LIN {X 0.040,Y -180.708,Z 1755.470,A 0.000,B 0.000,C 90.000,E1 264.552} C_DIS
LIN {X -0.041,Y -178.793,Z 1755.442,A 0.000,B 0.000,C 90.000,E1 259.511} C_DIS
LIN {X 0.037,Y -175.839,Z 1755.413,A 0.000,B 0.000,C 90.000,E1 254.393} C_DIS
LIN {X 0.036,Y -172.030,Z 1755.385,A 0.000,B 0.000,C 90.000,E1 249.263} C_DIS
LIN {X 0.012,Y -171.457,Z 1755.380,A 0.000,B 0.000,C 90.000,E1 248.411} C_DIS
LIN {X -0.008,Y -167.690,Z 1755.356,A 0.000,B 0.000,C 90.000,E1 244.101} C_DIS
LIN {X 0.006,Y -166.372,Z 1755.346,A 0.000,B 0.000,C 90.000,E1 242.359} C_DIS
LIN {X -0.001,Y -163.102,Z 1755.327,A 0.000,B 0.000,C 90.000,E1 238.869} C_DIS
LIN {X 0.048,Y -161.048,Z 1755.312,A 0.000,B 0.000,C 90.000,E1 236.215} C_DIS
LIN {X 0.033,Y -157.785,Z 1755.293,A 0.000,B 0.000,C 90.000,E1 232.683} C_DIS
LIN {X -0.024,Y -155.821,Z 1755.278,A 0.000,B 0.000,C 90.000,E1 230.033} C_DIS
LIN {X -0.067,Y -152.073,Z 1755.253,A 0.000,B 0.000,C 90.000,E1 225.567} C_DIS
LIN {X -0.048,Y -150.322,Z 1755.238,A 0.000,B 0.000,C 90.000,E1 222.852} C_DIS
LIN {X -0.026,Y -147.065,Z 1755.213,A 0.000,B 0.000,C 90.000,E1 218.302} C_DIS
LIN {X 0.081,Y -145.640,Z 1755.198,A 0.000,B 0.000,C 90.000,E1 215.518} C_DIS
LIN {X 0.079,Y -143.023,Z 1755.172,A 0.000,B 0.000,C 90.000,E1 210.924} C_DIS
LIN {X 0.010,Y -141.649,Z 1755.151,A 0.000,B 0.000,C 90.000,E1 207.257} C_DIS
LIN {X 0.060,Y -139.443,Z 1755.115,A 0.000,B 0.000,C 90.000,E1 200.737} C_DIS
LIN {X -0.018,Y -139.175,Z 1755.105,A 0.000,B 0.000,C 90.000,E1 198.906} C_DIS
LIN {X 0.010,Y -138.319,Z 1755.053,A 0.000,B 0.000,C 90.000,E1 189.557} C_DIS
LIN {X 0.019,Y -139.469,Z 1755.006,A 0.000,B 0.000,C 90.000,E1 181.146} C_DIS
LIN {X -0.040,Y -141.038,Z 1754.975,A 0.000,B 0.000,C 90.000,E1 175.584} C_DIS
LIN {X 0.055,Y -142.406,Z 1754.960,A 0.000,B 0.000,C 90.000,E1 172.761} C_DIS
LIN {X -0.024,Y -144.639,Z 1754.934,A 0.000,B 0.000,C 90.000,E1 168.173} C_DIS
LIN {X 0.036,Y -147.835,Z 1754.909,A 0.000,B 0.000,C 90.000,E1 163.559} C_DIS
LIN {X -0.020,Y -150.531,Z 1754.888,A 0.000,B 0.000,C 90.000,E1 159.934} C_DIS
LIN {X -0.001,Y -153.994,Z 1754.868,A 0.000,B 0.000,C 90.000,E1 156.305} C_DIS
LIN {X -0.080,Y -157.408,Z 1754.848,A 0.000,B 0.000,C 90.000,E1 152.743} C_DIS
LIN {X -0.001,Y -161.616,Z 1754.829,A 0.000,B 0.000,C 90.000,E1 149.154} C_DIS
LIN {X 0.101,Y -165.813,Z 1754.809,A 0.000,B 0.000,C 90.000,E1 145.595} C_DIS
LIN {X -0.011,Y -170.780,Z 1754.790,A 0.000,B 0.000,C 90.000,E1 142.145} C_DIS
LIN {X 0.012,Y -175.651,Z 1754.771,A 0.000,B 0.000,C 90.000,E1 138.690} C_DIS
LIN {X 0.009,Y -181.266,Z 1754.752,A 0.000,B 0.000,C 90.000,E1 135.283} C_DIS
LIN {X 0.009,Y -186.740,Z 1754.733,A 0.000,B 0.000,C 90.000,E1 131.919} C_DIS
LIN {X -0.039,Y -191.336,Z 1754.719,A 0.000,B 0.000,C 90.000,E1 129.439} C_DIS
LIN {X 0.007,Y -197.170,Z 1754.701,A 0.000,B 0.000,C 90.000,E1 126.137} C_DIS
LIN {X -0.075,Y -200.448,Z 1754.692,A 0.000,B 0.000,C 90.000,E1 124.532} C_DIS
LIN {X 0.108,Y -206.331,Z 1754.674,A 0.000,B 0.000,C 90.000,E1 121.258} C_DIS
LIN {X 0.076,Y -210.527,Z 1754.662,A 0.000,B 0.000,C 90.000,E1 119.205} C_DIS
LIN {X 0.072,Y -336.076,Z 1754.662,A 0.000,B 0.000,C 90.000,E1 119.205} C_DIS
LIN {X -0.025,Y -337.451,Z 1754.662,A 0.000,B 0.000,C 90.000,E1 119.205} C_DIS
LIN {X -0.160,Y -341.637,Z 1754.661,A 0.000,B 0.000,C 90.000,E1 119.077} C_DIS
LIN {X 0.005,Y -343.914,Z 1754.661,A 0.000,B 0.000,C 90.000,E1 118.899} C_DIS
LIN {X 0.117,Y -347.777,Z 1754.658,A 0.000,B 0.000,C 90.000,E1 118.487} C_DIS
LIN {X -0.014,Y -349.661,Z 1754.657,A 0.000,B 0.000,C 90.000,E1 118.231} C_DIS
LIN {X 0.039,Y -352.528,Z 1754.654,A 0.000,B 0.000,C 90.000,E1 117.641} C_DIS
LIN {X -0.051,Y -365.817,Z 1754.639,A 0.000,B 0.000,C 90.000,E1 114.951} C_DIS
LIN {X 0.124,Y -380.655,Z 1754.624,A 0.000,B 0.000,C 90.000,E1 112.280} C_DIS
LIN {X 0.058,Y -395.252,Z 1754.611,A 0.000,B 0.000,C 90.000,E1 109.993} C_DIS
LIN {X -0.057,Y -411.275,Z 1754.599,A 0.000,B 0.000,C 90.000,E1 107.764} C_DIS
LIN {X 0.109,Y -428.838,Z 1754.586,A 0.000,B 0.000,C 90.000,E1 105.552} C_DIS
LIN {X 0.213,Y -448.012,Z 1754.575,A 0.000,B 0.000,C 90.000,E1 103.411} C_DIS
LIN {X -0.213,Y -468.079,Z 1754.564,A 0.000,B 0.000,C 90.000,E1 101.478} C_DIS
LIN {X 0.253,Y -491.305,Z 1754.552,A 0.000,B 0.000,C 90.000,E1 99.378} C_DIS
LIN {X -0.047,Y -509.698,Z 1754.544,A 0.000,B 0.000,C 90.000,E1 97.936} C_DIS
LIN {X 0.195,Y -512.101,Z 1754.543,A 0.000,B 0.000,C 90.000,E1 97.701} C_DIS
LIN {X -0.240,Y -513.995,Z 1754.542,A 0.000,B 0.000,C 90.000,E1 97.530} C_DIS
LIN {X -0.100,Y -515.433,Z 1754.541,A 0.000,B 0.000,C 90.000,E1 97.296} C_DIS
LIN {X -0.240,Y -517.449,Z 1754.538,A 0.000,B 0.000,C 90.000,E1 96.834} C_DIS
LIN {X 0.143,Y -518.273,Z 1754.535,A 0.000,B 0.000,C 90.000,E1 96.315} C_DIS
LIN {X 0.022,Y -518.062,Z 1754.532,A 0.000,B 0.000,C 90.000,E1 95.853} C_DIS
LIN {X -0.097,Y -516.785,Z 1754.530,A 0.000,B 0.000,C 90.000,E1 95.391} C_DIS
LIN {X -0.179,Y -515.682,Z 1754.529,A 0.000,B 0.000,C 90.000,E1 95.163} C_DIS
LIN {X 0.206,Y -512.472,Z 1754.526,A 0.000,B 0.000,C 90.000,E1 94.645} C_DIS
LIN {X -0.042,Y -498.764,Z 1754.515,A 0.000,B 0.000,C 90.000,E1 92.751} C_DIS
LIN {X -0.166,Y -489.865,Z 1754.509,A 0.000,B 0.000,C 90.000,E1 91.547} C_DIS
LIN {X 0.038,Y -475.234,Z 1754.497,A 0.000,B 0.000,C 90.000,E1 89.542} C_DIS
LIN {X -0.133,Y -464.235,Z 1754.489,A 0.000,B 0.000,C 90.000,E1 88.051} C_DIS
LIN {X -0.045,Y -449.558,Z 1754.478,A 0.000,B 0.000,C 90.000,E1 85.988} C_DIS
LIN {X 0.029,Y -436.773,Z 1754.468,A 0.000,B 0.000,C 90.000,E1 84.147} C_DIS
LIN {X 0.170,Y -420.678,Z 1754.454,A 0.000,B 0.000,C 90.000,E1 81.724} C_DIS
LIN {X 0.111,Y -403.545,Z 1754.439,A 0.000,B 0.000,C 90.000,E1 78.993} C_DIS
LIN {X 0.190,Y -387.313,Z 1754.423,A 0.000,B 0.000,C 90.000,E1 76.172} C_DIS
LIN {X -0.120,Y -374.927,Z 1754.411,A 0.000,B 0.000,C 90.000,E1 73.921} C_DIS
LIN {X -0.149,Y -362.921,Z 1754.398,A 0.000,B 0.000,C 90.000,E1 71.583} C_DIS
LIN {X 0.096,Y -351.274,Z 1754.384,A 0.000,B 0.000,C 90.000,E1 69.156} C_DIS
LIN {X 0.118,Y -337.342,Z 1754.367,A 0.000,B 0.000,C 90.000,E1 66.102} C_DIS
LIN {X -0.021,Y -327.838,Z 1754.355,A 0.000,B 0.000,C 90.000,E1 63.948} C_DIS
LIN {X 0.149,Y -317.156,Z 1754.341,A 0.000,B 0.000,C 90.000,E1 61.385} C_DIS
LIN {X 0.069,Y -310.275,Z 1754.332,A 0.000,B 0.000,C 90.000,E1 59.793} C_DIS
LIN {X -0.116,Y -303.074,Z 1754.323,A 0.000,B 0.000,C 90.000,E1 58.201} C_DIS
LIN {X 0.091,Y -291.430,Z 1754.308,A 0.000,B 0.000,C 90.000,E1 55.515} C_DIS
LIN {X -0.022,Y -281.370,Z 1754.295,A 0.000,B 0.000,C 90.000,E1 53.176} C_DIS
LIN {X -0.088,Y -270.159,Z 1754.280,A 0.000,B 0.000,C 90.000,E1 50.436} C_DIS
LIN {X -0.127,Y -259.442,Z 1754.265,A 0.000,B 0.000,C 90.000,E1 47.634} C_DIS
LIN {X -0.123,Y -251.556,Z 1754.253,A 0.000,B 0.000,C 90.000,E1 45.486} C_DIS
LIN {X 0.050,Y -240.177,Z 1754.234,A 0.000,B 0.000,C 90.000,E1 42.162} C_DIS
LIN {X -0.059,Y -229.392,Z 1754.216,A 0.000,B 0.000,C 90.000,E1 38.830} C_DIS
LIN {X 0.037,Y -220.401,Z 1754.199,A 0.000,B 0.000,C 90.000,E1 35.758} C_DIS
LIN {X -0.010,Y -214.074,Z 1754.186,A 0.000,B 0.000,C 90.000,E1 33.452} C_DIS
LIN {X -0.091,Y -206.447,Z 1754.168,A 0.000,B 0.000,C 90.000,E1 30.335} C_DIS
LIN {X -0.035,Y -199.500,Z 1754.151,A 0.000,B 0.000,C 90.000,E1 27.129} C_DIS
LIN {X -0.065,Y -193.231,Z 1754.133,A 0.000,B 0.000,C 90.000,E1 23.898} C_DIS
LIN {X -0.047,Y -187.807,Z 1754.114,A 0.000,B 0.000,C 90.000,E1 20.610} C_DIS
LIN {X -0.012,Y -183.120,Z 1754.096,A 0.000,B 0.000,C 90.000,E1 17.275} C_DIS
LIN {X 0.093,Y -179.345,Z 1754.077,A 0.000,B 0.000,C 90.000,E1 13.883} C_DIS
LIN {X 0.020,Y -175.766,Z 1754.054,A 0.000,B 0.000,C 90.000,E1 9.670} C_DIS
LIN {X 0.052,Y -172.721,Z 1754.025,A 0.000,B 0.000,C 90.000,E1 4.531} C_DIS
LIN {X -0.052,Y -171.069,Z 1753.983,A 0.000,B 0.000,C 90.000,E1 356.963} C_DIS
LIN {X -0.058,Y -171.916,Z 1753.935,A 0.000,B 0.000,C 90.000,E1 348.342} C_DIS
LIN {X -0.011,Y -174.125,Z 1753.902,A 0.000,B 0.000,C 90.000,E1 342.308} C_DIS
LIN {X -0.005,Y -177.557,Z 1753.873,A 0.000,B 0.000,C 90.000,E1 337.177} C_DIS
LIN {X 0.041,Y -181.260,Z 1753.850,A 0.000,B 0.000,C 90.000,E1 332.922} C_DIS
LIN {X -0.056,Y -184.980,Z 1753.831,A 0.000,B 0.000,C 90.000,E1 329.587} C_DIS
LIN {X 0.061,Y -189.516,Z 1753.812,A 0.000,B 0.000,C 90.000,E1 326.215} C_DIS
LIN {X 0.027,Y -195.012,Z 1753.794,A 0.000,B 0.000,C 90.000,E1 322.924} C_DIS
LIN {X 0.007,Y -199.781,Z 1753.781,A 0.000,B 0.000,C 90.000,E1 320.481} C_DIS
LIN {X 0.088,Y -206.288,Z 1753.765,A 0.000,B 0.000,C 90.000,E1 317.634} C_DIS
LIN {X 0.112,Y -212.607,Z 1753.751,A 0.000,B 0.000,C 90.000,E1 315.243} C_DIS
LIN {X 0.048,Y -218.582,Z 1753.741,A 0.000,B 0.000,C 90.000,E1 313.299} C_DIS
LIN {X -0.061,Y -225.378,Z 1753.730,A 0.000,B 0.000,C 90.000,E1 311.391} C_DIS
LIN {X -0.016,Y -231.515,Z 1753.721,A 0.000,B 0.000,C 90.000,E1 309.850} C_DIS
LIN {X -0.007,Y -238.420,Z 1753.713,A 0.000,B 0.000,C 90.000,E1 308.338} C_DIS
LIN {X 0.089,Y -250.033,Z 1753.701,A 0.000,B 0.000,C 90.000,E1 306.091} C_DIS
LIN {X 0.078,Y -260.616,Z 1753.691,A 0.000,B 0.000,C 90.000,E1 304.278} C_DIS
LIN {X 0.027,Y -279.018,Z 1753.675,A 0.000,B 0.000,C 90.000,E1 301.465} C_DIS
LIN {X 0.018,Y -296.314,Z 1753.661,A 0.000,B 0.000,C 90.000,E1 299.077} C_DIS
LIN {X 0.108,Y -314.364,Z 1753.649,A 0.000,B 0.000,C 90.000,E1 296.744} C_DIS
LIN {X -0.008,Y -330.250,Z 1753.638,A 0.000,B 0.000,C 90.000,E1 294.847} C_DIS
LIN {X 0.141,Y -343.384,Z 1753.629,A 0.000,B 0.000,C 90.000,E1 293.259} C_DIS
LIN {X -0.111,Y -356.226,Z 1753.621,A 0.000,B 0.000,C 90.000,E1 291.770} C_DIS
LIN {X -0.037,Y -366.016,Z 1753.614,A 0.000,B 0.000,C 90.000,E1 290.556} C_DIS
LIN {X 0.204,Y -372.830,Z 1753.609,A 0.000,B 0.000,C 90.000,E1 289.631} C_DIS
LIN {X 0.024,Y -378.910,Z 1753.604,A 0.000,B 0.000,C 90.000,E1 288.779} C_DIS
LIN {X 0.136,Y -382.533,Z 1753.601,A 0.000,B 0.000,C 90.000,E1 288.181} C_DIS
LIN {X -0.091,Y -385.669,Z 1753.598,A 0.000,B 0.000,C 90.000,E1 287.638} C_DIS
LIN {X 0.069,Y -388.324,Z 1753.595,A 0.000,B 0.000,C 90.000,E1 287.040} C_DIS
LIN {X -0.124,Y -390.623,Z 1753.592,A 0.000,B 0.000,C 90.000,E1 286.496} C_DIS
LIN {X 0.070,Y -392.522,Z 1753.588,A 0.000,B 0.000,C 90.000,E1 285.898} C_DIS
LIN {X -0.215,Y -394.106,Z 1753.585,A 0.000,B 0.000,C 90.000,E1 285.371} C_DIS
LIN {X -0.002,Y -395.323,Z 1753.582,A 0.000,B 0.000,C 90.000,E1 284.773} C_DIS
LIN {X 0.123,Y -396.187,Z 1753.579,A 0.000,B 0.000,C 90.000,E1 284.189} C_DIS
LIN {X -0.034,Y -396.671,Z 1753.576,A 0.000,B 0.000,C 90.000,E1 283.647} C_DIS
LIN {X 0.105,Y -396.800,Z 1753.573,A 0.000,B 0.000,C 90.000,E1 283.063} C_DIS
LIN {X -0.138,Y -396.538,Z 1753.570,A 0.000,B 0.000,C 90.000,E1 282.535} C_DIS
LIN {X 0.008,Y -395.863,Z 1753.566,A 0.000,B 0.000,C 90.000,E1 281.951} C_DIS
LIN {X 0.152,Y -394.688,Z 1753.563,A 0.000,B 0.000,C 90.000,E1 281.366} C_DIS
LIN {X -0.095,Y -393.020,Z 1753.560,A 0.000,B 0.000,C 90.000,E1 280.838} C_DIS
LIN {X 0.037,Y -390.808,Z 1753.557,A 0.000,B 0.000,C 90.000,E1 280.254} C_DIS
LIN {X 0.149,Y -388.030,Z 1753.554,A 0.000,B 0.000,C 90.000,E1 279.670} C_DIS
LIN {X -0.037,Y -380.278,Z 1753.546,A 0.000,B 0.000,C 90.000,E1 278.276} C_DIS
LIN {X 0.025,Y -375.925,Z 1753.541,A 0.000,B 0.000,C 90.000,E1 277.409} C_DIS
LIN {X -0.008,Y -372.510,Z 1753.538,A 0.000,B 0.000,C 90.000,E1 276.834} C_DIS
LIN {X -0.058,Y -368.487,Z 1753.535,A 0.000,B 0.000,C 90.000,E1 276.258} C_DIS
LIN {X -0.127,Y -363.774,Z 1753.531,A 0.000,B 0.000,C 90.000,E1 275.682} C_DIS
LIN {X 0.136,Y -358.283,Z 1753.528,A 0.000,B 0.000,C 90.000,E1 275.049} C_DIS
LIN {X -0.072,Y -352.446,Z 1753.525,A 0.000,B 0.000,C 90.000,E1 274.531} C_DIS
LIN {X -0.027,Y -346.500,Z 1753.522,A 0.000,B 0.000,C 90.000,E1 274.012} C_DIS
LIN {X 0.160,Y -340.378,Z 1753.520,A 0.000,B 0.000,C 90.000,E1 273.498} C_DIS
LIN {X 0.024,Y -330.914,Z 1753.516,A 0.000,B 0.000,C 90.000,E1 272.865} C_DIS
LIN {X 0.057,Y -324.422,Z 1753.514,A 0.000,B 0.000,C 90.000,E1 272.465} C_DIS
LIN {X -0.040,Y -317.608,Z 1753.512,A 0.000,B 0.000,C 90.000,E1 272.121} C_DIS
LIN {X 0.117,Y -310.610,Z 1753.510,A 0.000,B 0.000,C 90.000,E1 271.776} C_DIS
LIN {X -0.078,Y -303.341,Z 1753.509,A 0.000,B 0.000,C 90.000,E1 271.547} C_DIS
LIN {X 0.069,Y -292.260,Z 1753.507,A 0.000,B 0.000,C 90.000,E1 271.203} C_DIS
LIN {X 0.001,Y -281.588,Z 1753.505,A 0.000,B 0.000,C 90.000,E1 270.974} C_DIS
LIN {X -0.106,Y -273.354,Z 1753.505,A 0.000,B 0.000,C 90.000,E1 270.859} C_DIS
LIN {X -0.092,Y -258.515,Z 1753.504,A 0.000,B 0.000,C 90.000,E1 270.688} C_DIS
LIN {X 0.031,Y -239.967,Z 1753.503,A 0.000,B 0.000,C 90.000,E1 270.516} C_DIS
LIN {X -0.015,Y -237.145,Z 1753.503,A 0.000,B 0.000,C 90.000,E1 270.516} C_DIS
LIN {X -0.047,Y -181.565,Z 1753.503,A 0.000,B 0.000,C 90.000,E1 270.516} C_DIS
LIN {X 0.054,Y -181.117,Z 1753.489,A 0.000,B 0.000,C 90.000,E1 267.936} C_DIS
LIN {X 0.042,Y -180.906,Z 1753.475,A 0.000,B 0.000,C 90.000,E1 265.412} C_DIS
LIN {X -0.081,Y -180.716,Z 1753.470,A 0.000,B 0.000,C 90.000,E1 264.609} C_DIS
LIN {X 0.017,Y -178.804,Z 1753.442,A 0.000,B 0.000,C 90.000,E1 259.511} C_DIS
LIN {X 0.093,Y -175.848,Z 1753.413,A 0.000,B 0.000,C 90.000,E1 254.393} C_DIS
LIN {X 0.053,Y -172.584,Z 1753.390,A 0.000,B 0.000,C 90.000,E1 250.134} C_DIS
LIN {X 0.069,Y -171.474,Z 1753.380,A 0.000,B 0.000,C 90.000,E1 248.411} C_DIS
LIN {X 0.048,Y -167.704,Z 1753.356,A 0.000,B 0.000,C 90.000,E1 244.101} C_DIS
LIN {X 0.061,Y -166.391,Z 1753.347,A 0.000,B 0.000,C 90.000,E1 242.359} C_DIS
LIN {X 0.052,Y -163.118,Z 1753.327,A 0.000,B 0.000,C 90.000,E1 238.869} C_DIS
LIN {X 0.102,Y -161.067,Z 1753.313,A 0.000,B 0.000,C 90.000,E1 236.215} C_DIS
LIN {X -0.010,Y -157.800,Z 1753.293,A 0.000,B 0.000,C 90.000,E1 232.718} C_DIS
LIN {X -0.072,Y -155.836,Z 1753.278,A 0.000,B 0.000,C 90.000,E1 230.070} C_DIS
LIN {X -0.015,Y -152.086,Z 1753.253,A 0.000,B 0.000,C 90.000,E1 225.567} C_DIS
LIN {X 0.004,Y -150.337,Z 1753.238,A 0.000,B 0.000,C 90.000,E1 222.852} C_DIS
LIN {X 0.025,Y -147.076,Z 1753.213,A 0.000,B 0.000,C 90.000,E1 218.302} C_DIS
LIN {X -0.071,Y -145.650,Z 1753.198,A 0.000,B 0.000,C 90.000,E1 215.598} C_DIS
LIN {X -0.067,Y -143.032,Z 1753.172,A 0.000,B 0.000,C 90.000,E1 211.003} C_DIS
LIN {X 0.059,Y -141.657,Z 1753.152,A 0.000,B 0.000,C 90.000,E1 207.257} C_DIS
LIN {X -0.022,Y -139.447,Z 1753.115,A 0.000,B 0.000,C 90.000,E1 200.791} C_DIS
LIN {X 0.031,Y -139.180,Z 1753.105,A 0.000,B 0.000,C 90.000,E1 198.906} C_DIS
LIN {X 0.059,Y -138.320,Z 1753.053,A 0.000,B 0.000,C 90.000,E1 189.557} C_DIS
LIN {X 0.069,Y -139.465,Z 1753.006,A 0.000,B 0.000,C 90.000,E1 181.146} C_DIS
LIN {X 0.010,Y -141.029,Z 1752.975,A 0.000,B 0.000,C 90.000,E1 175.584} C_DIS
LIN {X -0.036,Y -142.396,Z 1752.960,A 0.000,B 0.000,C 90.000,E1 172.818} C_DIS
LIN {X 0.026,Y -144.628,Z 1752.934,A 0.000,B 0.000,C 90.000,E1 168.173} C_DIS
LIN {X -0.055,Y -147.823,Z 1752.909,A 0.000,B 0.000,C 90.000,E1 163.614} C_DIS
LIN {X 0.031,Y -150.514,Z 1752.889,A 0.000,B 0.000,C 90.000,E1 159.934} C_DIS
LIN {X 0.052,Y -153.976,Z 1752.868,A 0.000,B 0.000,C 90.000,E1 156.305} C_DIS
LIN {X -0.027,Y -157.387,Z 1752.849,A 0.000,B 0.000,C 90.000,E1 152.743} C_DIS
LIN {X -0.085,Y -161.592,Z 1752.829,A 0.000,B 0.000,C 90.000,E1 149.203} C_DIS
LIN {X -0.075,Y -165.789,Z 1752.809,A 0.000,B 0.000,C 90.000,E1 145.674} C_DIS
LIN {X -0.089,Y -170.750,Z 1752.790,A 0.000,B 0.000,C 90.000,E1 142.190} C_DIS
LIN {X 0.069,Y -175.622,Z 1752.771,A 0.000,B 0.000,C 90.000,E1 138.690} C_DIS
LIN {X -0.062,Y -181.238,Z 1752.752,A 0.000,B 0.000,C 90.000,E1 135.324} C_DIS
LIN {X 0.069,Y -186.708,Z 1752.733,A 0.000,B 0.000,C 90.000,E1 131.919} C_DIS
LIN {X 0.021,Y -191.307,Z 1752.719,A 0.000,B 0.000,C 90.000,E1 129.439} C_DIS
LIN {X -0.048,Y -197.136,Z 1752.701,A 0.000,B 0.000,C 90.000,E1 126.171} C_DIS
LIN {X -0.013,Y -200.413,Z 1752.692,A 0.000,B 0.000,C 90.000,E1 124.532} C_DIS
LIN {X -0.112,Y -206.297,Z 1752.674,A 0.000,B 0.000,C 90.000,E1 121.337} C_DIS
LIN {X -0.118,Y -210.483,Z 1752.662,A 0.000,B 0.000,C 90.000,E1 119.283} C_DIS
LIN {X -0.072,Y -335.448,Z 1752.662,A 0.000,B 0.000,C 90.000,E1 119.255} C_DIS
LIN {X 0.077,Y -337.648,Z 1752.662,A 0.000,B 0.000,C 90.000,E1 119.205} C_DIS
LIN {X -0.056,Y -341.622,Z 1752.661,A 0.000,B 0.000,C 90.000,E1 119.077} C_DIS
LIN {X -0.193,Y -343.865,Z 1752.661,A 0.000,B 0.000,C 90.000,E1 118.949} C_DIS
LIN {X 0.190,Y -347.733,Z 1752.658,A 0.000,B 0.000,C 90.000,E1 118.487} C_DIS
LIN {X 0.047,Y -349.612,Z 1752.657,A 0.000,B 0.000,C 90.000,E1 118.231} C_DIS
LIN {X 0.087,Y -352.470,Z 1752.654,A 0.000,B 0.000,C 90.000,E1 117.641} C_DIS
LIN {X -0.004,Y -365.755,Z 1752.639,A 0.000,B 0.000,C 90.000,E1 114.951} C_DIS
LIN {X -0.181,Y -380.588,Z 1752.624,A 0.000,B 0.000,C 90.000,E1 112.333} C_DIS
LIN {X 0.106,Y -395.180,Z 1752.611,A 0.000,B 0.000,C 90.000,E1 109.993} C_DIS
LIN {X -0.009,Y -411.199,Z 1752.599,A 0.000,B 0.000,C 90.000,E1 107.764} C_DIS
LIN {X 0.157,Y -428.756,Z 1752.587,A 0.000,B 0.000,C 90.000,E1 105.552} C_DIS
LIN {X 0.260,Y -447.927,Z 1752.575,A 0.000,B 0.000,C 90.000,E1 103.411} C_DIS
LIN {X -0.169,Y -467.992,Z 1752.564,A 0.000,B 0.000,C 90.000,E1 101.478} C_DIS
LIN {X -0.189,Y -491.216,Z 1752.552,A 0.000,B 0.000,C 90.000,E1 99.434} C_DIS
LIN {X 0.117,Y -509.660,Z 1752.544,A 0.000,B 0.000,C 90.000,E1 97.936} C_DIS
LIN {X -0.095,Y -512.041,Z 1752.543,A 0.000,B 0.000,C 90.000,E1 97.757} C_DIS
LIN {X 0.169,Y -515.407,Z 1752.541,A 0.000,B 0.000,C 90.000,E1 97.296} C_DIS
LIN {X 0.062,Y -516.621,Z 1752.539,A 0.000,B 0.000,C 90.000,E1 97.068} C_DIS
LIN {X 0.019,Y -517.495,Z 1752.538,A 0.000,B 0.000,C 90.000,E1 96.834} C_DIS
LIN {X -0.106,Y -518.377,Z 1752.535,A 0.000,B 0.000,C 90.000,E1 96.372} C_DIS
LIN {X -0.228,Y -518.230,Z 1752.533,A 0.000,B 0.000,C 90.000,E1 95.910} C_DIS
LIN {X 0.169,Y -517.031,Z 1752.530,A 0.000,B 0.000,C 90.000,E1 95.391} C_DIS
LIN {X 0.086,Y -515.979,Z 1752.529,A 0.000,B 0.000,C 90.000,E1 95.163} C_DIS
LIN {X 0.004,Y -514.554,Z 1752.527,A 0.000,B 0.000,C 90.000,E1 94.935} C_DIS
LIN {X -0.159,Y -500.528,Z 1752.517,A 0.000,B 0.000,C 90.000,E1 93.037} C_DIS
LIN {X 0.228,Y -491.573,Z 1752.510,A 0.000,B 0.000,C 90.000,E1 91.776} C_DIS
LIN {X -0.021,Y -476.875,Z 1752.499,A 0.000,B 0.000,C 90.000,E1 89.828} C_DIS
LIN {X -0.177,Y -465.908,Z 1752.491,A 0.000,B 0.000,C 90.000,E1 88.339} C_DIS
LIN {X 0.205,Y -453.040,Z 1752.481,A 0.000,B 0.000,C 90.000,E1 86.502} C_DIS
LIN {X -0.127,Y -440.253,Z 1752.471,A 0.000,B 0.000,C 90.000,E1 84.723} C_DIS
LIN {X 0.112,Y -424.031,Z 1752.457,A 0.000,B 0.000,C 90.000,E1 82.299} C_DIS
LIN {X -0.202,Y -405.029,Z 1752.441,A 0.000,B 0.000,C 90.000,E1 79.342} C_DIS
LIN {X -0.008,Y -387.125,Z 1752.423,A 0.000,B 0.000,C 90.000,E1 76.228} C_DIS
LIN {X 0.048,Y -374.724,Z 1752.411,A 0.000,B 0.000,C 90.000,E1 73.921} C_DIS
LIN {X 0.009,Y -362.673,Z 1752.398,A 0.000,B 0.000,C 90.000,E1 71.583} C_DIS
LIN {X -0.047,Y -349.566,Z 1752.383,A 0.000,B 0.000,C 90.000,E1 68.901} C_DIS
LIN {X -0.063,Y -335.711,Z 1752.366,A 0.000,B 0.000,C 90.000,E1 65.845} C_DIS
LIN {X 0.023,Y -324.836,Z 1752.352,A 0.000,B 0.000,C 90.000,E1 63.332} C_DIS
LIN {X -0.091,Y -315.496,Z 1752.339,A 0.000,B 0.000,C 90.000,E1 61.129} C_DIS
LIN {X 0.069,Y -308.534,Z 1752.331,A 0.000,B 0.000,C 90.000,E1 59.488} C_DIS
LIN {X 0.039,Y -299.832,Z 1752.320,A 0.000,B 0.000,C 90.000,E1 57.533} C_DIS
LIN {X -0.068,Y -289.739,Z 1752.307,A 0.000,B 0.000,C 90.000,E1 55.229} C_DIS
LIN {X 0.010,Y -279.690,Z 1752.294,A 0.000,B 0.000,C 90.000,E1 52.844} C_DIS
LIN {X -0.020,Y -269.921,Z 1752.280,A 0.000,B 0.000,C 90.000,E1 50.436} C_DIS
LIN {X -0.068,Y -259.180,Z 1752.265,A 0.000,B 0.000,C 90.000,E1 47.634} C_DIS
LIN {X -0.071,Y -251.282,Z 1752.253,A 0.000,B 0.000,C 90.000,E1 45.486} C_DIS
LIN {X -0.086,Y -239.872,Z 1752.234,A 0.000,B 0.000,C 90.000,E1 42.204} C_DIS
LIN {X -0.026,Y -229.083,Z 1752.216,A 0.000,B 0.000,C 90.000,E1 38.830} C_DIS
LIN {X -0.118,Y -220.083,Z 1752.199,A 0.000,B 0.000,C 90.000,E1 35.804} C_DIS
LIN {X -0.001,Y -211.822,Z 1752.182,A 0.000,B 0.000,C 90.000,E1 32.673} C_DIS
LIN {X -0.071,Y -204.405,Z 1752.164,A 0.000,B 0.000,C 90.000,E1 29.539} C_DIS
LIN {X 0.018,Y -197.626,Z 1752.146,A 0.000,B 0.000,C 90.000,E1 26.309} C_DIS
LIN {X -0.067,Y -193.019,Z 1752.133,A 0.000,B 0.000,C 90.000,E1 23.898} C_DIS
LIN {X -0.055,Y -187.617,Z 1752.114,A 0.000,B 0.000,C 90.000,E1 20.610} C_DIS
LIN {X -0.024,Y -182.937,Z 1752.096,A 0.000,B 0.000,C 90.000,E1 17.275} C_DIS
LIN {X 0.077,Y -179.158,Z 1752.077,A 0.000,B 0.000,C 90.000,E1 13.883} C_DIS
LIN {X -0.002,Y -175.557,Z 1752.054,A 0.000,B 0.000,C 90.000,E1 9.670} C_DIS
LIN {X 0.023,Y -172.524,Z 1752.025,A 0.000,B 0.000,C 90.000,E1 4.531} C_DIS
LIN {X -0.056,Y -170.849,Z 1751.983,A 0.000,B 0.000,C 90.000,E1 356.963} C_DIS
LIN {X 0.094,Y -171.687,Z 1751.935,A 0.000,B 0.000,C 90.000,E1 348.285} C_DIS
LIN {X -0.037,Y -173.908,Z 1751.902,A 0.000,B 0.000,C 90.000,E1 342.308} C_DIS
LIN {X -0.040,Y -177.365,Z 1751.873,A 0.000,B 0.000,C 90.000,E1 337.177} C_DIS
LIN {X -0.001,Y -181.113,Z 1751.850,A 0.000,B 0.000,C 90.000,E1 332.922} C_DIS
LIN {X 0.059,Y -184.870,Z 1751.831,A 0.000,B 0.000,C 90.000,E1 329.537} C_DIS
LIN {X 0.012,Y -189.465,Z 1751.812,A 0.000,B 0.000,C 90.000,E1 326.215} C_DIS
LIN {X -0.025,Y -194.988,Z 1751.794,A 0.000,B 0.000,C 90.000,E1 322.924} C_DIS
LIN {X 0.107,Y -199.822,Z 1751.780,A 0.000,B 0.000,C 90.000,E1 320.436} C_DIS
LIN {X 0.034,Y -206.384,Z 1751.765,A 0.000,B 0.000,C 90.000,E1 317.634} C_DIS
LIN {X 0.058,Y -212.736,Z 1751.751,A 0.000,B 0.000,C 90.000,E1 315.243} C_DIS
LIN {X -0.005,Y -218.767,Z 1751.741,A 0.000,B 0.000,C 90.000,E1 313.299} C_DIS
LIN {X 0.035,Y -225.601,Z 1751.730,A 0.000,B 0.000,C 90.000,E1 311.353} C_DIS
LIN {X -0.066,Y -231.770,Z 1751.721,A 0.000,B 0.000,C 90.000,E1 309.850} C_DIS
LIN {X 0.059,Y -240.572,Z 1751.711,A 0.000,B 0.000,C 90.000,E1 307.935} C_DIS
LIN {X 0.044,Y -250.331,Z 1751.701,A 0.000,B 0.000,C 90.000,E1 306.091} C_DIS
LIN {X 0.074,Y -263.146,Z 1751.688,A 0.000,B 0.000,C 90.000,E1 303.913} C_DIS
LIN {X -0.010,Y -279.290,Z 1751.675,A 0.000,B 0.000,C 90.000,E1 301.465} C_DIS
LIN {X -0.015,Y -296.556,Z 1751.661,A 0.000,B 0.000,C 90.000,E1 299.077} C_DIS
LIN {X 0.079,Y -314.647,Z 1751.649,A 0.000,B 0.000,C 90.000,E1 296.744} C_DIS
LIN {X -0.044,Y -330.537,Z 1751.638,A 0.000,B 0.000,C 90.000,E1 294.847} C_DIS
LIN {X 0.125,Y -343.659,Z 1751.629,A 0.000,B 0.000,C 90.000,E1 293.259} C_DIS
LIN {X -0.121,Y -356.503,Z 1751.621,A 0.000,B 0.000,C 90.000,E1 291.770} C_DIS
LIN {X -0.044,Y -366.294,Z 1751.614,A 0.000,B 0.000,C 90.000,E1 290.556} C_DIS
LIN {X 0.200,Y -373.112,Z 1751.609,A 0.000,B 0.000,C 90.000,E1 289.631} C_DIS
LIN {X 0.022,Y -379.215,Z 1751.604,A 0.000,B 0.000,C 90.000,E1 288.779} C_DIS
LIN {X 0.136,Y -382.821,Z 1751.601,A 0.000,B 0.000,C 90.000,E1 288.181} C_DIS
LIN {X 0.049,Y -387.390,Z 1751.596,A 0.000,B 0.000,C 90.000,E1 287.330} C_DIS
LIN {X -0.119,Y -390.954,Z 1751.592,A 0.000,B 0.000,C 90.000,E1 286.496} C_DIS
LIN {X 0.077,Y -392.796,Z 1751.588,A 0.000,B 0.000,C 90.000,E1 285.898} C_DIS
LIN {X -0.205,Y -394.441,Z 1751.585,A 0.000,B 0.000,C 90.000,E1 285.371} C_DIS
LIN {X 0.010,Y -395.640,Z 1751.582,A 0.000,B 0.000,C 90.000,E1 284.773} C_DIS
LIN {X 0.135,Y -396.508,Z 1751.579,A 0.000,B 0.000,C 90.000,E1 284.189} C_DIS
LIN {X -0.019,Y -396.982,Z 1751.576,A 0.000,B 0.000,C 90.000,E1 283.647} C_DIS
LIN {X 0.122,Y -397.114,Z 1751.573,A 0.000,B 0.000,C 90.000,E1 283.063} C_DIS
LIN {X -0.119,Y -396.870,Z 1751.570,A 0.000,B 0.000,C 90.000,E1 282.535} C_DIS
LIN {X 0.028,Y -396.155,Z 1751.566,A 0.000,B 0.000,C 90.000,E1 281.951} C_DIS
LIN {X -0.212,Y -394.938,Z 1751.563,A 0.000,B 0.000,C 90.000,E1 281.422} C_DIS
LIN {X -0.071,Y -393.289,Z 1751.560,A 0.000,B 0.000,C 90.000,E1 280.838} C_DIS
LIN {X 0.062,Y -391.042,Z 1751.557,A 0.000,B 0.000,C 90.000,E1 280.254} C_DIS
LIN {X 0.176,Y -388.182,Z 1751.554,A 0.000,B 0.000,C 90.000,E1 279.670} C_DIS
LIN {X -0.093,Y -381.743,Z 1751.547,A 0.000,B 0.000,C 90.000,E1 278.568} C_DIS
LIN {X -0.017,Y -375.972,Z 1751.541,A 0.000,B 0.000,C 90.000,E1 277.409} C_DIS
LIN {X -0.050,Y -372.546,Z 1751.538,A 0.000,B 0.000,C 90.000,E1 276.834} C_DIS
LIN {X -0.099,Y -368.517,Z 1751.535,A 0.000,B 0.000,C 90.000,E1 276.258} C_DIS
LIN {X -0.168,Y -363.735,Z 1751.531,A 0.000,B 0.000,C 90.000,E1 275.682} C_DIS
LIN {X 0.097,Y -358.236,Z 1751.528,A 0.000,B 0.000,C 90.000,E1 275.049} C_DIS
LIN {X -0.109,Y -352.361,Z 1751.525,A 0.000,B 0.000,C 90.000,E1 274.531} C_DIS
LIN {X -0.108,Y -343.415,Z 1751.521,A 0.000,B 0.000,C 90.000,E1 273.784} C_DIS
LIN {X -0.143,Y -337.243,Z 1751.518,A 0.000,B 0.000,C 90.000,E1 273.326} C_DIS
LIN {X 0.046,Y -330.881,Z 1751.516,A 0.000,B 0.000,C 90.000,E1 272.865} C_DIS
LIN {X 0.098,Y -324.460,Z 1751.514,A 0.000,B 0.000,C 90.000,E1 272.465} C_DIS
LIN {X 0.037,Y -317.651,Z 1751.512,A 0.000,B 0.000,C 90.000,E1 272.121} C_DIS
LIN {X -0.108,Y -310.696,Z 1751.510,A 0.000,B 0.000,C 90.000,E1 271.835} C_DIS
LIN {X 0.007,Y -303.420,Z 1751.509,A 0.000,B 0.000,C 90.000,E1 271.547} C_DIS
LIN {X -0.143,Y -292.357,Z 1751.507,A 0.000,B 0.000,C 90.000,E1 271.260} C_DIS
LIN {X 0.068,Y -281.518,Z 1751.505,A 0.000,B 0.000,C 90.000,E1 270.974} C_DIS
LIN {X -0.053,Y -272.881,Z 1751.505,A 0.000,B 0.000,C 90.000,E1 270.859} C_DIS
LIN {X -0.038,Y -257.820,Z 1751.504,A 0.000,B 0.000,C 90.000,E1 270.688} C_DIS
LIN {X -0.066,Y -242.724,Z 1751.503,A 0.000,B 0.000,C 90.000,E1 270.573} C_DIS
LIN {X 0.026,Y -232.060,Z 1751.503,A 0.000,B 0.000,C 90.000,E1 270.516} C_DIS
LIN {X 0.001,Y -181.562,Z 1751.503,A 0.000,B 0.000,C 90.000,E1 270.516} C_DIS
LIN {X 0.020,Y -181.276,Z 1751.493,A 0.000,B 0.000,C 90.000,E1 268.797} C_DIS
LIN {X 0.068,Y -180.906,Z 1751.475,A 0.000,B 0.000,C 90.000,E1 265.412} C_DIS
LIN {X -0.056,Y -180.720,Z 1751.470,A 0.000,B 0.000,C 90.000,E1 264.609} C_DIS
LIN {X 0.042,Y -178.807,Z 1751.442,A 0.000,B 0.000,C 90.000,E1 259.511} C_DIS
LIN {X -0.051,Y -175.853,Z 1751.413,A 0.000,B 0.000,C 90.000,E1 254.448} C_DIS
LIN {X -0.069,Y -173.179,Z 1751.395,A 0.000,B 0.000,C 90.000,E1 251.040} C_DIS
LIN {X -0.066,Y -171.480,Z 1751.380,A 0.000,B 0.000,C 90.000,E1 248.465} C_DIS
LIN {X -0.079,Y -167.711,Z 1751.356,A 0.000,B 0.000,C 90.000,E1 244.152} C_DIS
LIN {X -0.062,Y -166.399,Z 1751.347,A 0.000,B 0.000,C 90.000,E1 242.410} C_DIS
LIN {X 0.076,Y -163.124,Z 1751.327,A 0.000,B 0.000,C 90.000,E1 238.869} C_DIS
LIN {X -0.098,Y -161.076,Z 1751.313,A 0.000,B 0.000,C 90.000,E1 236.294} C_DIS
LIN {X 0.013,Y -157.807,Z 1751.293,A 0.000,B 0.000,C 90.000,E1 232.718} C_DIS
LIN {X -0.048,Y -155.842,Z 1751.278,A 0.000,B 0.000,C 90.000,E1 230.070} C_DIS
LIN {X 0.008,Y -152.093,Z 1751.253,A 0.000,B 0.000,C 90.000,E1 225.567} C_DIS
LIN {X 0.027,Y -150.344,Z 1751.238,A 0.000,B 0.000,C 90.000,E1 222.852} C_DIS
LIN {X 0.047,Y -147.082,Z 1751.213,A 0.000,B 0.000,C 90.000,E1 218.302} C_DIS
LIN {X -0.049,Y -145.655,Z 1751.198,A 0.000,B 0.000,C 90.000,E1 215.598} C_DIS
LIN {X -0.045,Y -143.037,Z 1751.172,A 0.000,B 0.000,C 90.000,E1 211.003} C_DIS
LIN {X 0.081,Y -141.661,Z 1751.152,A 0.000,B 0.000,C 90.000,E1 207.257} C_DIS
LIN {X 0.000,Y -139.448,Z 1751.115,A 0.000,B 0.000,C 90.000,E1 200.791} C_DIS
LIN {X 0.053,Y -139.182,Z 1751.105,A 0.000,B 0.000,C 90.000,E1 198.906} C_DIS
LIN {X -0.055,Y -138.321,Z 1751.053,A 0.000,B 0.000,C 90.000,E1 189.613} C_DIS
LIN {X -0.049,Y -139.464,Z 1751.007,A 0.000,B 0.000,C 90.000,E1 181.203} C_DIS
LIN {X 0.031,Y -141.025,Z 1750.976,A 0.000,B 0.000,C 90.000,E1 175.584} C_DIS
LIN {X -0.013,Y -142.391,Z 1750.960,A 0.000,B 0.000,C 90.000,E1 172.818} C_DIS
LIN {X 0.049,Y -144.622,Z 1750.934,A 0.000,B 0.000,C 90.000,E1 168.173} C_DIS
LIN {X -0.032,Y -147.817,Z 1750.909,A 0.000,B 0.000,C 90.000,E1 163.614} C_DIS
LIN {X 0.054,Y -150.507,Z 1750.889,A 0.000,B 0.000,C 90.000,E1 159.934} C_DIS
LIN {X -0.066,Y -153.966,Z 1750.869,A 0.000,B 0.000,C 90.000,E1 156.357} C_DIS
LIN {X -0.003,Y -157.378,Z 1750.849,A 0.000,B 0.000,C 90.000,E1 152.743} C_DIS
LIN {X -0.062,Y -161.580,Z 1750.829,A 0.000,B 0.000,C 90.000,E1 149.203} C_DIS
LIN {X -0.050,Y -165.777,Z 1750.809,A 0.000,B 0.000,C 90.000,E1 145.674} C_DIS
LIN {X -0.065,Y -170.738,Z 1750.790,A 0.000,B 0.000,C 90.000,E1 142.190} C_DIS
LIN {X -0.022,Y -175.610,Z 1750.771,A 0.000,B 0.000,C 90.000,E1 138.728} C_DIS
LIN {X -0.036,Y -181.226,Z 1750.752,A 0.000,B 0.000,C 90.000,E1 135.324} C_DIS
LIN {X 0.095,Y -186.693,Z 1750.733,A 0.000,B 0.000,C 90.000,E1 131.919} C_DIS
LIN {X 0.047,Y -191.294,Z 1750.719,A 0.000,B 0.000,C 90.000,E1 129.439} C_DIS
LIN {X -0.021,Y -197.121,Z 1750.701,A 0.000,B 0.000,C 90.000,E1 126.171} C_DIS
LIN {X 0.015,Y -200.397,Z 1750.692,A 0.000,B 0.000,C 90.000,E1 124.532} C_DIS
LIN {X -0.084,Y -206.281,Z 1750.674,A 0.000,B 0.000,C 90.000,E1 121.337} C_DIS
LIN {X -0.055,Y -210.454,Z 1750.663,A 0.000,B 0.000,C 90.000,E1 119.283} C_DIS
LIN {X -0.143,Y -336.326,Z 1750.663,A 0.000,B 0.000,C 90.000,E1 119.283} C_DIS
LIN {X 0.087,Y -341.468,Z 1750.662,A 0.000,B 0.000,C 90.000,E1 119.077} C_DIS
LIN {X -0.147,Y -343.929,Z 1750.661,A 0.000,B 0.000,C 90.000,E1 118.949} C_DIS
LIN {X 0.211,Y -347.755,Z 1750.658,A 0.000,B 0.000,C 90.000,E1 118.487} C_DIS
LIN {X 0.042,Y -349.625,Z 1750.657,A 0.000,B 0.000,C 90.000,E1 118.231} C_DIS
LIN {X 0.076,Y -353.877,Z 1750.652,A 0.000,B 0.000,C 90.000,E1 117.334} C_DIS
LIN {X 0.037,Y -367.327,Z 1750.637,A 0.000,B 0.000,C 90.000,E1 114.643} C_DIS
LIN {X -0.094,Y -382.347,Z 1750.622,A 0.000,B 0.000,C 90.000,E1 112.025} C_DIS
LIN {X 0.106,Y -397.115,Z 1750.609,A 0.000,B 0.000,C 90.000,E1 109.704} C_DIS
LIN {X 0.174,Y -413.324,Z 1750.597,A 0.000,B 0.000,C 90.000,E1 107.457} C_DIS
LIN {X -0.022,Y -431.085,Z 1750.585,A 0.000,B 0.000,C 90.000,E1 105.300} C_DIS
LIN {X 0.044,Y -450.436,Z 1750.573,A 0.000,B 0.000,C 90.000,E1 103.175} C_DIS
LIN {X 0.238,Y -470.573,Z 1750.562,A 0.000,B 0.000,C 90.000,E1 101.186} C_DIS
LIN {X -0.127,Y -493.840,Z 1750.551,A 0.000,B 0.000,C 90.000,E1 99.208} C_DIS
LIN {X 0.080,Y -509.686,Z 1750.544,A 0.000,B 0.000,C 90.000,E1 97.936} C_DIS
LIN {X -0.131,Y -512.018,Z 1750.543,A 0.000,B 0.000,C 90.000,E1 97.757} C_DIS
LIN {X -0.059,Y -513.919,Z 1750.542,A 0.000,B 0.000,C 90.000,E1 97.530} C_DIS
LIN {X 0.081,Y -515.373,Z 1750.541,A 0.000,B 0.000,C 90.000,E1 97.296} C_DIS
LIN {X -0.021,Y -516.568,Z 1750.539,A 0.000,B 0.000,C 90.000,E1 97.068} C_DIS
LIN {X -0.059,Y -517.430,Z 1750.538,A 0.000,B 0.000,C 90.000,E1 96.834} C_DIS
LIN {X -0.185,Y -518.297,Z 1750.535,A 0.000,B 0.000,C 90.000,E1 96.372} C_DIS
LIN {X 0.208,Y -518.129,Z 1750.533,A 0.000,B 0.000,C 90.000,E1 95.853} C_DIS
LIN {X 0.090,Y -516.904,Z 1750.530,A 0.000,B 0.000,C 90.000,E1 95.391} C_DIS
LIN {X 0.007,Y -515.834,Z 1750.529,A 0.000,B 0.000,C 90.000,E1 95.163} C_DIS
LIN {X -0.074,Y -514.383,Z 1750.527,A 0.000,B 0.000,C 90.000,E1 94.935} C_DIS
LIN {X 0.137,Y -498.315,Z 1750.515,A 0.000,B 0.000,C 90.000,E1 92.751} C_DIS
LIN {X -0.140,Y -487.414,Z 1750.507,A 0.000,B 0.000,C 90.000,E1 91.318} C_DIS
LIN {X 0.008,Y -472.780,Z 1750.496,A 0.000,B 0.000,C 90.000,E1 89.312} C_DIS
LIN {X 0.050,Y -459.913,Z 1750.486,A 0.000,B 0.000,C 90.000,E1 87.535} C_DIS
LIN {X 0.057,Y -445.272,Z 1750.475,A 0.000,B 0.000,C 90.000,E1 85.469} C_DIS
LIN {X -0.189,Y -430.719,Z 1750.463,A 0.000,B 0.000,C 90.000,E1 83.394} C_DIS
LIN {X 0.137,Y -416.522,Z 1750.451,A 0.000,B 0.000,C 90.000,E1 81.197} C_DIS
LIN {X -0.030,Y -399.551,Z 1750.436,A 0.000,B 0.000,C 90.000,E1 78.465} C_DIS
LIN {X -0.060,Y -383.532,Z 1750.420,A 0.000,B 0.000,C 90.000,E1 75.644} C_DIS
LIN {X 0.008,Y -371.221,Z 1750.407,A 0.000,B 0.000,C 90.000,E1 73.323} C_DIS
LIN {X -0.054,Y -357.756,Z 1750.393,A 0.000,B 0.000,C 90.000,E1 70.678} C_DIS
LIN {X -0.094,Y -343.422,Z 1750.376,A 0.000,B 0.000,C 90.000,E1 67.667} C_DIS
LIN {X 0.047,Y -332.464,Z 1750.362,A 0.000,B 0.000,C 90.000,E1 65.177} C_DIS
LIN {X 0.039,Y -321.617,Z 1750.348,A 0.000,B 0.000,C 90.000,E1 62.666} C_DIS
LIN {X 0.069,Y -313.588,Z 1750.338,A 0.000,B 0.000,C 90.000,E1 60.745} C_DIS
LIN {X -0.026,Y -305.104,Z 1750.327,A 0.000,B 0.000,C 90.000,E1 58.820} C_DIS
LIN {X 0.057,Y -294.955,Z 1750.314,A 0.000,B 0.000,C 90.000,E1 56.501} C_DIS
LIN {X 0.104,Y -286.362,Z 1750.303,A 0.000,B 0.000,C 90.000,E1 54.482} C_DIS
LIN {X -0.017,Y -275.013,Z 1750.288,A 0.000,B 0.000,C 90.000,E1 51.778} C_DIS
LIN {X -0.054,Y -262.691,Z 1750.270,A 0.000,B 0.000,C 90.000,E1 48.647} C_DIS
LIN {X 0.037,Y -253.410,Z 1750.256,A 0.000,B 0.000,C 90.000,E1 46.134} C_DIS
LIN {X 0.086,Y -243.097,Z 1750.240,A 0.000,B 0.000,C 90.000,E1 43.218} C_DIS
LIN {X 0.047,Y -232.112,Z 1750.222,A 0.000,B 0.000,C 90.000,E1 39.886} C_DIS
LIN {X -0.075,Y -221.780,Z 1750.203,A 0.000,B 0.000,C 90.000,E1 36.503} C_DIS
LIN {X 0.079,Y -213.360,Z 1750.186,A 0.000,B 0.000,C 90.000,E1 33.372} C_DIS
LIN {X -0.026,Y -205.761,Z 1750.168,A 0.000,B 0.000,C 90.000,E1 30.256} C_DIS
LIN {X 0.052,Y -197.269,Z 1750.146,A 0.000,B 0.000,C 90.000,E1 26.232} C_DIS
LIN {X -0.037,Y -191.283,Z 1750.128,A 0.000,B 0.000,C 90.000,E1 23.003} C_DIS
LIN {X 0.029,Y -186.088,Z 1750.109,A 0.000,B 0.000,C 90.000,E1 19.685} C_DIS
LIN {X -0.041,Y -181.652,Z 1750.091,A 0.000,B 0.000,C 90.000,E1 16.370} C_DIS
LIN {X -0.061,Y -178.114,Z 1750.072,A 0.000,B 0.000,C 90.000,E1 13.008} C_DIS
LIN {X -0.023,Y -174.728,Z 1750.049,A 0.000,B 0.000,C 90.000,E1 8.746} C_DIS
LIN {X -0.040,Y -171.943,Z 1750.020,A 0.000,B 0.000,C 90.000,E1 3.612} C_DIS
LIN {X -0.067,Y -170.589,Z 1749.978,A 0.000,B 0.000,C 90.000,E1 356.102} C_DIS
LIN {X 0.077,Y -171.454,Z 1749.935,A 0.000,B 0.000,C 90.000,E1 348.285} C_DIS
LIN {X -0.063,Y -173.702,Z 1749.902,A 0.000,B 0.000,C 90.000,E1 342.308} C_DIS
LIN {X 0.096,Y -176.533,Z 1749.878,A 0.000,B 0.000,C 90.000,E1 337.975} C_DIS
LIN {X -0.040,Y -180.145,Z 1749.854,A 0.000,B 0.000,C 90.000,E1 333.768} C_DIS
LIN {X 0.014,Y -184.779,Z 1749.831,A 0.000,B 0.000,C 90.000,E1 329.537} C_DIS
LIN {X -0.035,Y -189.399,Z 1749.812,A 0.000,B 0.000,C 90.000,E1 326.215} C_DIS
LIN {X -0.075,Y -194.966,Z 1749.794,A 0.000,B 0.000,C 90.000,E1 322.924} C_DIS
LIN {X 0.055,Y -199.865,Z 1749.780,A 0.000,B 0.000,C 90.000,E1 320.436} C_DIS
LIN {X -0.019,Y -206.468,Z 1749.765,A 0.000,B 0.000,C 90.000,E1 317.634} C_DIS
LIN {X 0.006,Y -212.874,Z 1749.751,A 0.000,B 0.000,C 90.000,E1 315.243} C_DIS
LIN {X -0.056,Y -218.950,Z 1749.740,A 0.000,B 0.000,C 90.000,E1 313.299} C_DIS
LIN {X -0.015,Y -225.827,Z 1749.730,A 0.000,B 0.000,C 90.000,E1 311.353} C_DIS
LIN {X 0.064,Y -232.046,Z 1749.721,A 0.000,B 0.000,C 90.000,E1 309.806} C_DIS
LIN {X 0.046,Y -239.000,Z 1749.713,A 0.000,B 0.000,C 90.000,E1 308.302} C_DIS
LIN {X 0.001,Y -250.622,Z 1749.701,A 0.000,B 0.000,C 90.000,E1 306.091} C_DIS
LIN {X -0.022,Y -267.908,Z 1749.684,A 0.000,B 0.000,C 90.000,E1 303.214} C_DIS
LIN {X 0.052,Y -286.821,Z 1749.669,A 0.000,B 0.000,C 90.000,E1 300.413} C_DIS
LIN {X 0.076,Y -304.492,Z 1749.656,A 0.000,B 0.000,C 90.000,E1 298.052} C_DIS
LIN {X -0.029,Y -322.834,Z 1749.643,A 0.000,B 0.000,C 90.000,E1 295.796} C_DIS
LIN {X 0.029,Y -336.066,Z 1749.635,A 0.000,B 0.000,C 90.000,E1 294.207} C_DIS
LIN {X 0.115,Y -346.489,Z 1749.628,A 0.000,B 0.000,C 90.000,E1 292.950} C_DIS
LIN {X -0.131,Y -356.770,Z 1749.621,A 0.000,B 0.000,C 90.000,E1 291.770} C_DIS
LIN {X -0.052,Y -366.564,Z 1749.614,A 0.000,B 0.000,C 90.000,E1 290.556} C_DIS
LIN {X 0.196,Y -373.387,Z 1749.609,A 0.000,B 0.000,C 90.000,E1 289.631} C_DIS
LIN {X 0.019,Y -379.483,Z 1749.604,A 0.000,B 0.000,C 90.000,E1 288.779} C_DIS
LIN {X 0.136,Y -383.100,Z 1749.601,A 0.000,B 0.000,C 90.000,E1 288.181} C_DIS
LIN {X -0.088,Y -386.274,Z 1749.598,A 0.000,B 0.000,C 90.000,E1 287.638} C_DIS
LIN {X 0.076,Y -388.984,Z 1749.595,A 0.000,B 0.000,C 90.000,E1 287.040} C_DIS
LIN {X -0.115,Y -391.268,Z 1749.592,A 0.000,B 0.000,C 90.000,E1 286.496} C_DIS
LIN {X 0.083,Y -393.172,Z 1749.588,A 0.000,B 0.000,C 90.000,E1 285.898} C_DIS
LIN {X -0.197,Y -394.729,Z 1749.585,A 0.000,B 0.000,C 90.000,E1 285.371} C_DIS
LIN {X 0.021,Y -395.968,Z 1749.582,A 0.000,B 0.000,C 90.000,E1 284.773} C_DIS
LIN {X 0.149,Y -396.810,Z 1749.579,A 0.000,B 0.000,C 90.000,E1 284.189} C_DIS
LIN {X -0.005,Y -397.305,Z 1749.576,A 0.000,B 0.000,C 90.000,E1 283.647} C_DIS
LIN {X 0.138,Y -397.444,Z 1749.573,A 0.000,B 0.000,C 90.000,E1 283.063} C_DIS
LIN {X -0.101,Y -397.168,Z 1749.570,A 0.000,B 0.000,C 90.000,E1 282.535} C_DIS
LIN {X 0.048,Y -396.475,Z 1749.566,A 0.000,B 0.000,C 90.000,E1 281.951} C_DIS
LIN {X -0.191,Y -395.272,Z 1749.563,A 0.000,B 0.000,C 90.000,E1 281.422} C_DIS
LIN {X -0.047,Y -393.572,Z 1749.560,A 0.000,B 0.000,C 90.000,E1 280.838} C_DIS
LIN {X 0.088,Y -391.266,Z 1749.557,A 0.000,B 0.000,C 90.000,E1 280.254} C_DIS
LIN {X -0.131,Y -386.778,Z 1749.552,A 0.000,B 0.000,C 90.000,E1 279.434} C_DIS
LIN {X -0.064,Y -381.830,Z 1749.547,A 0.000,B 0.000,C 90.000,E1 278.568} C_DIS
LIN {X 0.018,Y -376.388,Z 1749.542,A 0.000,B 0.000,C 90.000,E1 277.466} C_DIS
LIN {X -0.012,Y -373.078,Z 1749.538,A 0.000,B 0.000,C 90.000,E1 276.891} C_DIS
LIN {X -0.059,Y -369.077,Z 1749.535,A 0.000,B 0.000,C 90.000,E1 276.315} C_DIS
LIN {X -0.126,Y -364.308,Z 1749.532,A 0.000,B 0.000,C 90.000,E1 275.739} C_DIS
LIN {X 0.141,Y -358.879,Z 1749.528,A 0.000,B 0.000,C 90.000,E1 275.106} C_DIS
LIN {X -0.092,Y -353.038,Z 1749.525,A 0.000,B 0.000,C 90.000,E1 274.588} C_DIS
LIN {X -0.157,Y -343.974,Z 1749.521,A 0.000,B 0.000,C 90.000,E1 273.841} C_DIS
LIN {X 0.160,Y -337.877,Z 1749.519,A 0.000,B 0.000,C 90.000,E1 273.326} C_DIS
LIN {X -0.006,Y -331.533,Z 1749.516,A 0.000,B 0.000,C 90.000,E1 272.922} C_DIS
LIN {X 0.023,Y -325.096,Z 1749.514,A 0.000,B 0.000,C 90.000,E1 272.522} C_DIS
LIN {X -0.038,Y -318.365,Z 1749.512,A 0.000,B 0.000,C 90.000,E1 272.178} C_DIS
LIN {X 0.131,Y -311.405,Z 1749.510,A 0.000,B 0.000,C 90.000,E1 271.835} C_DIS
LIN {X -0.126,Y -300.384,Z 1749.508,A 0.000,B 0.000,C 90.000,E1 271.489} C_DIS
LIN {X 0.123,Y -289.261,Z 1749.506,A 0.000,B 0.000,C 90.000,E1 271.146} C_DIS
LIN {X -0.125,Y -281.648,Z 1749.506,A 0.000,B 0.000,C 90.000,E1 271.031} C_DIS
LIN {X 0.019,Y -272.814,Z 1749.505,A 0.000,B 0.000,C 90.000,E1 270.859} C_DIS
LIN {X 0.036,Y -257.569,Z 1749.504,A 0.000,B 0.000,C 90.000,E1 270.688} C_DIS
LIN {X 0.004,Y -242.974,Z 1749.503,A 0.000,B 0.000,C 90.000,E1 270.573} C_DIS
LIN {X 0.093,Y -233.403,Z 1749.503,A 0.000,B 0.000,C 90.000,E1 270.516} C_DIS
LIN {X 0.054,Y -181.560,Z 1749.503,A 0.000,B 0.000,C 90.000,E1 270.516} C_DIS
LIN {X 0.072,Y -181.279,Z 1749.493,A 0.000,B 0.000,C 90.000,E1 268.797} C_DIS
LIN {X -0.060,Y -180.907,Z 1749.475,A 0.000,B 0.000,C 90.000,E1 265.469} C_DIS
LIN {X -0.003,Y -180.728,Z 1749.470,A 0.000,B 0.000,C 90.000,E1 264.609} C_DIS
LIN {X 0.095,Y -178.817,Z 1749.442,A 0.000,B 0.000,C 90.000,E1 259.511} C_DIS
LIN {X 0.001,Y -175.861,Z 1749.414,A 0.000,B 0.000,C 90.000,E1 254.448} C_DIS
LIN {X 0.050,Y -173.827,Z 1749.399,A 0.000,B 0.000,C 90.000,E1 251.873} C_DIS
LIN {X -0.016,Y -171.495,Z 1749.380,A 0.000,B 0.000,C 90.000,E1 248.465} C_DIS
LIN {X -0.028,Y -167.724,Z 1749.356,A 0.000,B 0.000,C 90.000,E1 244.152} C_DIS
LIN {X -0.012,Y -166.417,Z 1749.347,A 0.000,B 0.000,C 90.000,E1 242.410} C_DIS
LIN {X -0.014,Y -163.139,Z 1749.327,A 0.000,B 0.000,C 90.000,E1 238.918} C_DIS
LIN {X -0.048,Y -161.093,Z 1749.313,A 0.000,B 0.000,C 90.000,E1 236.294} C_DIS
LIN {X -0.064,Y -157.822,Z 1749.293,A 0.000,B 0.000,C 90.000,E1 232.763} C_DIS
LIN {X 0.000,Y -155.856,Z 1749.278,A 0.000,B 0.000,C 90.000,E1 230.070} C_DIS
LIN {X 0.055,Y -152.105,Z 1749.253,A 0.000,B 0.000,C 90.000,E1 225.567} C_DIS
LIN {X 0.074,Y -150.356,Z 1749.238,A 0.000,B 0.000,C 90.000,E1 222.852} C_DIS
LIN {X 0.002,Y -147.092,Z 1749.213,A 0.000,B 0.000,C 90.000,E1 218.338} C_DIS
LIN {X -0.003,Y -145.663,Z 1749.198,A 0.000,B 0.000,C 90.000,E1 215.598} C_DIS
LIN {X 0.001,Y -143.045,Z 1749.172,A 0.000,B 0.000,C 90.000,E1 211.003} C_DIS
LIN {X 0.001,Y -141.669,Z 1749.152,A 0.000,B 0.000,C 90.000,E1 207.308} C_DIS
LIN {X 0.046,Y -139.452,Z 1749.116,A 0.000,B 0.000,C 90.000,E1 200.791} C_DIS
LIN {X -0.034,Y -139.186,Z 1749.105,A 0.000,B 0.000,C 90.000,E1 198.960} C_DIS
LIN {X -0.011,Y -138.321,Z 1749.053,A 0.000,B 0.000,C 90.000,E1 189.613} C_DIS
LIN {X -0.003,Y -139.461,Z 1749.007,A 0.000,B 0.000,C 90.000,E1 181.203} C_DIS
LIN {X -0.064,Y -141.018,Z 1748.976,A 0.000,B 0.000,C 90.000,E1 175.641} C_DIS
LIN {X 0.026,Y -142.772,Z 1748.955,A 0.000,B 0.000,C 90.000,E1 171.894} C_DIS
LIN {X 0.013,Y -145.184,Z 1748.929,A 0.000,B 0.000,C 90.000,E1 167.285} C_DIS
LIN {X 0.015,Y -147.805,Z 1748.909,A 0.000,B 0.000,C 90.000,E1 163.614} C_DIS
LIN {X -0.091,Y -150.491,Z 1748.889,A 0.000,B 0.000,C 90.000,E1 160.007} C_DIS
LIN {X -0.018,Y -153.949,Z 1748.869,A 0.000,B 0.000,C 90.000,E1 156.357} C_DIS
LIN {X 0.045,Y -157.359,Z 1748.849,A 0.000,B 0.000,C 90.000,E1 152.743} C_DIS
LIN {X -0.011,Y -161.557,Z 1748.829,A 0.000,B 0.000,C 90.000,E1 149.203} C_DIS
LIN {X 0.000,Y -165.755,Z 1748.809,A 0.000,B 0.000,C 90.000,E1 145.674} C_DIS
LIN {X -0.013,Y -170.711,Z 1748.790,A 0.000,B 0.000,C 90.000,E1 142.190} C_DIS
LIN {X 0.030,Y -175.584,Z 1748.771,A 0.000,B 0.000,C 90.000,E1 138.728} C_DIS
LIN {X 0.018,Y -181.201,Z 1748.752,A 0.000,B 0.000,C 90.000,E1 135.324} C_DIS
LIN {X 0.010,Y -186.664,Z 1748.733,A 0.000,B 0.000,C 90.000,E1 131.962} C_DIS
LIN {X -0.045,Y -191.268,Z 1748.719,A 0.000,B 0.000,C 90.000,E1 129.483} C_DIS
LIN {X 0.035,Y -197.090,Z 1748.701,A 0.000,B 0.000,C 90.000,E1 126.171} C_DIS
LIN {X 0.072,Y -200.364,Z 1748.692,A 0.000,B 0.000,C 90.000,E1 124.532} C_DIS
LIN {X -0.027,Y -206.250,Z 1748.674,A 0.000,B 0.000,C 90.000,E1 121.337} C_DIS
LIN {X 0.036,Y -210.409,Z 1748.663,A 0.000,B 0.000,C 90.000,E1 119.283} C_DIS
LIN {X 0.004,Y -336.058,Z 1748.663,A 0.000,B 0.000,C 90.000,E1 119.283} C_DIS
LIN {X 0.182,Y -341.469,Z 1748.662,A 0.000,B 0.000,C 90.000,E1 119.077} C_DIS
LIN {X -0.052,Y -343.890,Z 1748.661,A 0.000,B 0.000,C 90.000,E1 118.949} C_DIS
LIN {X -0.033,Y -347.723,Z 1748.659,A 0.000,B 0.000,C 90.000,E1 118.537} C_DIS
LIN {X 0.087,Y -349.587,Z 1748.657,A 0.000,B 0.000,C 90.000,E1 118.231} C_DIS
LIN {X -0.016,Y -355.250,Z 1748.650,A 0.000,B 0.000,C 90.000,E1 117.052} C_DIS
LIN {X 0.144,Y -368.868,Z 1748.635,A 0.000,B 0.000,C 90.000,E1 114.335} C_DIS
LIN {X 0.067,Y -384.063,Z 1748.621,A 0.000,B 0.000,C 90.000,E1 111.716} C_DIS
LIN {X -0.058,Y -399.002,Z 1748.608,A 0.000,B 0.000,C 90.000,E1 109.450} C_DIS
LIN {X -0.083,Y -415.395,Z 1748.596,A 0.000,B 0.000,C 90.000,E1 107.221} C_DIS
LIN {X 0.182,Y -433.355,Z 1748.583,A 0.000,B 0.000,C 90.000,E1 105.009} C_DIS
LIN {X -0.064,Y -452.844,Z 1748.572,A 0.000,B 0.000,C 90.000,E1 102.939} C_DIS
LIN {X -0.175,Y -473.051,Z 1748.561,A 0.000,B 0.000,C 90.000,E1 101.007} C_DIS
LIN {X 0.076,Y -496.412,Z 1748.550,A 0.000,B 0.000,C 90.000,E1 98.973} C_DIS
LIN {X 0.103,Y -509.619,Z 1748.544,A 0.000,B 0.000,C 90.000,E1 97.936} C_DIS
LIN {X -0.108,Y -511.902,Z 1748.543,A 0.000,B 0.000,C 90.000,E1 97.757} C_DIS
LIN {X -0.063,Y -513.790,Z 1748.542,A 0.000,B 0.000,C 90.000,E1 97.530} C_DIS
LIN {X 0.050,Y -515.229,Z 1748.541,A 0.000,B 0.000,C 90.000,E1 97.296} C_DIS
LIN {X -0.091,Y -517.232,Z 1748.538,A 0.000,B 0.000,C 90.000,E1 96.834} C_DIS
LIN {X -0.224,Y -518.061,Z 1748.535,A 0.000,B 0.000,C 90.000,E1 96.372} C_DIS
LIN {X 0.168,Y -517.862,Z 1748.533,A 0.000,B 0.000,C 90.000,E1 95.853} C_DIS
LIN {X 0.049,Y -516.597,Z 1748.530,A 0.000,B 0.000,C 90.000,E1 95.391} C_DIS
LIN {X -0.034,Y -515.500,Z 1748.529,A 0.000,B 0.000,C 90.000,E1 95.163} C_DIS
LIN {X -0.117,Y -514.012,Z 1748.527,A 0.000,B 0.000,C 90.000,E1 94.935} C_DIS
LIN {X 0.086,Y -497.867,Z 1748.515,A 0.000,B 0.000,C 90.000,E1 92.751} C_DIS
LIN {X -0.196,Y -486.973,Z 1748.507,A 0.000,B 0.000,C 90.000,E1 91.318} C_DIS
LIN {X -0.057,Y -472.344,Z 1748.496,A 0.000,B 0.000,C 90.000,E1 89.312} C_DIS
LIN {X -0.022,Y -459.474,Z 1748.486,A 0.000,B 0.000,C 90.000,E1 87.535} C_DIS
LIN {X 0.226,Y -446.665,Z 1748.476,A 0.000,B 0.000,C 90.000,E1 85.698} C_DIS
LIN {X -0.039,Y -432.086,Z 1748.465,A 0.000,B 0.000,C 90.000,E1 83.628} C_DIS
LIN {X -0.106,Y -417.834,Z 1748.453,A 0.000,B 0.000,C 90.000,E1 81.489} C_DIS
LIN {X 0.164,Y -400.753,Z 1748.437,A 0.000,B 0.000,C 90.000,E1 78.701} C_DIS
LIN {X 0.159,Y -384.660,Z 1748.422,A 0.000,B 0.000,C 90.000,E1 75.880} C_DIS
LIN {X -0.110,Y -372.279,Z 1748.409,A 0.000,B 0.000,C 90.000,E1 73.614} C_DIS
LIN {X -0.125,Y -358.752,Z 1748.394,A 0.000,B 0.000,C 90.000,E1 70.967} C_DIS
LIN {X 0.072,Y -344.335,Z 1748.377,A 0.000,B 0.000,C 90.000,E1 67.922} C_DIS
LIN {X -0.077,Y -333.339,Z 1748.364,A 0.000,B 0.000,C 90.000,E1 65.485} C_DIS
LIN {X 0.084,Y -322.452,Z 1748.350,A 0.000,B 0.000,C 90.000,E1 62.948} C_DIS
LIN {X -0.001,Y -314.434,Z 1748.339,A 0.000,B 0.000,C 90.000,E1 61.051} C_DIS
LIN {X -0.122,Y -307.417,Z 1748.330,A 0.000,B 0.000,C 90.000,E1 59.459} C_DIS
LIN {X 0.115,Y -297.342,Z 1748.318,A 0.000,B 0.000,C 90.000,E1 57.120} C_DIS
LIN {X -0.050,Y -287.354,Z 1748.304,A 0.000,B 0.000,C 90.000,E1 54.815} C_DIS
LIN {X -0.023,Y -274.580,Z 1748.287,A 0.000,B 0.000,C 90.000,E1 51.743} C_DIS
LIN {X 0.076,Y -263.575,Z 1748.272,A 0.000,B 0.000,C 90.000,E1 48.933} C_DIS
LIN {X 0.007,Y -254.246,Z 1748.258,A 0.000,B 0.000,C 90.000,E1 46.458} C_DIS
LIN {X 0.077,Y -243.878,Z 1748.242,A 0.000,B 0.000,C 90.000,E1 43.542} C_DIS
LIN {X 0.039,Y -232.821,Z 1748.224,A 0.000,B 0.000,C 90.000,E1 40.216} C_DIS
LIN {X 0.102,Y -222.406,Z 1748.205,A 0.000,B 0.000,C 90.000,E1 36.790} C_DIS
LIN {X -0.006,Y -214.958,Z 1748.190,A 0.000,B 0.000,C 90.000,E1 34.119} C_DIS
LIN {X -0.070,Y -207.176,Z 1748.172,A 0.000,B 0.000,C 90.000,E1 31.003} C_DIS
LIN {X 0.101,Y -200.218,Z 1748.154,A 0.000,B 0.000,C 90.000,E1 27.769} C_DIS
LIN {X -0.092,Y -193.858,Z 1748.136,A 0.000,B 0.000,C 90.000,E1 24.591} C_DIS
LIN {X 0.013,Y -188.298,Z 1748.118,A 0.000,B 0.000,C 90.000,E1 21.280} C_DIS
LIN {X 0.060,Y -183.521,Z 1748.100,A 0.000,B 0.000,C 90.000,E1 17.946} C_DIS
LIN {X 0.052,Y -179.534,Z 1748.081,A 0.000,B 0.000,C 90.000,E1 14.592} C_DIS
LIN {X 0.019,Y -175.732,Z 1748.058,A 0.000,B 0.000,C 90.000,E1 10.366} C_DIS
LIN {X 0.069,Y -172.489,Z 1748.029,A 0.000,B 0.000,C 90.000,E1 5.220} C_DIS
LIN {X -0.049,Y -170.493,Z 1747.988,A 0.000,B 0.000,C 90.000,E1 357.822} C_DIS
LIN {X -0.031,Y -170.690,Z 1747.949,A 0.000,B 0.000,C 90.000,E1 350.905} C_DIS
LIN {X -0.023,Y -172.337,Z 1747.916,A 0.000,B 0.000,C 90.000,E1 344.866} C_DIS
LIN {X 0.022,Y -175.095,Z 1747.887,A 0.000,B 0.000,C 90.000,E1 339.699} C_DIS
LIN {X 0.024,Y -178.459,Z 1747.864,A 0.000,B 0.000,C 90.000,E1 335.433} C_DIS
LIN {X 0.097,Y -182.659,Z 1747.840,A 0.000,B 0.000,C 90.000,E1 331.179} C_DIS
LIN {X -0.039,Y -186.892,Z 1747.821,A 0.000,B 0.000,C 90.000,E1 327.867} C_DIS
LIN {X 0.017,Y -192.041,Z 1747.803,A 0.000,B 0.000,C 90.000,E1 324.529} C_DIS
LIN {X 0.013,Y -196.531,Z 1747.789,A 0.000,B 0.000,C 90.000,E1 322.065} C_DIS
LIN {X 0.017,Y -201.708,Z 1747.776,A 0.000,B 0.000,C 90.000,E1 319.622} C_DIS
LIN {X -0.003,Y -209.691,Z 1747.758,A 0.000,B 0.000,C 90.000,E1 316.419} C_DIS
LIN {X 0.092,Y -216.594,Z 1747.745,A 0.000,B 0.000,C 90.000,E1 314.028} C_DIS
LIN {X -0.061,Y -223.180,Z 1747.734,A 0.000,B 0.000,C 90.000,E1 312.123} C_DIS
LIN {X 0.129,Y -229.098,Z 1747.725,A 0.000,B 0.000,C 90.000,E1 310.539} C_DIS
LIN {X 0.034,Y -237.475,Z 1747.715,A 0.000,B 0.000,C 90.000,E1 308.669} C_DIS
LIN {X -0.042,Y -248.877,Z 1747.703,A 0.000,B 0.000,C 90.000,E1 306.457} C_DIS
LIN {X -0.110,Y -265.921,Z 1747.686,A 0.000,B 0.000,C 90.000,E1 303.579} C_DIS
LIN {X 0.058,Y -284.612,Z 1747.671,A 0.000,B 0.000,C 90.000,E1 300.747} C_DIS
LIN {X 0.047,Y -304.728,Z 1747.656,A 0.000,B 0.000,C 90.000,E1 298.052} C_DIS
LIN {X -0.084,Y -323.149,Z 1747.643,A 0.000,B 0.000,C 90.000,E1 295.796} C_DIS
LIN {X -0.036,Y -336.392,Z 1747.634,A 0.000,B 0.000,C 90.000,E1 294.207} C_DIS
LIN {X 0.051,Y -346.824,Z 1747.628,A 0.000,B 0.000,C 90.000,E1 292.950} C_DIS
LIN {X 0.138,Y -357.100,Z 1747.621,A 0.000,B 0.000,C 90.000,E1 291.716} C_DIS
LIN {X -0.111,Y -366.874,Z 1747.614,A 0.000,B 0.000,C 90.000,E1 290.556} C_DIS
LIN {X 0.137,Y -373.696,Z 1747.609,A 0.000,B 0.000,C 90.000,E1 289.631} C_DIS
LIN {X -0.142,Y -377.883,Z 1747.606,A 0.000,B 0.000,C 90.000,E1 289.087} C_DIS
LIN {X 0.081,Y -383.437,Z 1747.601,A 0.000,B 0.000,C 90.000,E1 288.181} C_DIS
LIN {X -0.142,Y -386.607,Z 1747.598,A 0.000,B 0.000,C 90.000,E1 287.638} C_DIS
LIN {X 0.025,Y -389.328,Z 1747.595,A 0.000,B 0.000,C 90.000,E1 287.040} C_DIS
LIN {X -0.165,Y -391.573,Z 1747.592,A 0.000,B 0.000,C 90.000,E1 286.496} C_DIS
LIN {X 0.035,Y -393.476,Z 1747.588,A 0.000,B 0.000,C 90.000,E1 285.898} C_DIS
LIN {X 0.138,Y -395.039,Z 1747.585,A 0.000,B 0.000,C 90.000,E1 285.315} C_DIS
LIN {X -0.024,Y -396.231,Z 1747.582,A 0.000,B 0.000,C 90.000,E1 284.773} C_DIS
LIN {X 0.105,Y -397.105,Z 1747.579,A 0.000,B 0.000,C 90.000,E1 284.189} C_DIS
LIN {X -0.046,Y -397.607,Z 1747.576,A 0.000,B 0.000,C 90.000,E1 283.647} C_DIS
LIN {X 0.098,Y -397.748,Z 1747.573,A 0.000,B 0.000,C 90.000,E1 283.063} C_DIS
LIN {X -0.140,Y -397.446,Z 1747.570,A 0.000,B 0.000,C 90.000,E1 282.535} C_DIS
LIN {X 0.013,Y -396.728,Z 1747.566,A 0.000,B 0.000,C 90.000,E1 281.951} C_DIS
LIN {X 0.162,Y -395.553,Z 1747.563,A 0.000,B 0.000,C 90.000,E1 281.366} C_DIS
LIN {X -0.079,Y -393.816,Z 1747.560,A 0.000,B 0.000,C 90.000,E1 280.838} C_DIS
LIN {X 0.058,Y -391.491,Z 1747.557,A 0.000,B 0.000,C 90.000,E1 280.254} C_DIS
LIN {X 0.174,Y -388.542,Z 1747.554,A 0.000,B 0.000,C 90.000,E1 279.670} C_DIS
LIN {X -0.091,Y -381.921,Z 1747.547,A 0.000,B 0.000,C 90.000,E1 278.568} C_DIS
LIN {X 0.034,Y -376.508,Z 1747.542,A 0.000,B 0.000,C 90.000,E1 277.466} C_DIS
LIN {X 0.003,Y -373.175,Z 1747.538,A 0.000,B 0.000,C 90.000,E1 276.891} C_DIS
LIN {X -0.043,Y -369.187,Z 1747.535,A 0.000,B 0.000,C 90.000,E1 276.315} C_DIS
LIN {X -0.110,Y -364.379,Z 1747.532,A 0.000,B 0.000,C 90.000,E1 275.739} C_DIS
LIN {X 0.158,Y -358.896,Z 1747.529,A 0.000,B 0.000,C 90.000,E1 275.106} C_DIS
LIN {X -0.080,Y -353.041,Z 1747.525,A 0.000,B 0.000,C 90.000,E1 274.588} C_DIS
LIN {X -0.101,Y -344.042,Z 1747.521,A 0.000,B 0.000,C 90.000,E1 273.841} C_DIS
LIN {X -0.112,Y -337.996,Z 1747.519,A 0.000,B 0.000,C 90.000,E1 273.383} C_DIS
LIN {X 0.087,Y -331.713,Z 1747.516,A 0.000,B 0.000,C 90.000,E1 272.922} C_DIS
LIN {X 0.142,Y -325.305,Z 1747.514,A 0.000,B 0.000,C 90.000,E1 272.522} C_DIS
LIN {X 0.081,Y -318.609,Z 1747.512,A 0.000,B 0.000,C 90.000,E1 272.178} C_DIS
LIN {X -0.058,Y -311.686,Z 1747.510,A 0.000,B 0.000,C 90.000,E1 271.892} C_DIS
LIN {X 0.051,Y -304.455,Z 1747.509,A 0.000,B 0.000,C 90.000,E1 271.604} C_DIS
LIN {X 0.073,Y -297.264,Z 1747.508,A 0.000,B 0.000,C 90.000,E1 271.375} C_DIS
LIN {X 0.128,Y -286.222,Z 1747.506,A 0.000,B 0.000,C 90.000,E1 271.088} C_DIS
LIN {X -0.048,Y -278.391,Z 1747.505,A 0.000,B 0.000,C 90.000,E1 270.974} C_DIS
LIN {X -0.102,Y -264.001,Z 1747.504,A 0.000,B 0.000,C 90.000,E1 270.802} C_DIS
LIN {X -0.116,Y -244.992,Z 1747.503,A 0.000,B 0.000,C 90.000,E1 270.630} C_DIS
LIN {X -0.070,Y -233.030,Z 1747.503,A 0.000,B 0.000,C 90.000,E1 270.573} C_DIS
LIN {X -0.074,Y -181.557,Z 1747.503,A 0.000,B 0.000,C 90.000,E1 270.573} C_DIS
LIN {X -0.024,Y -181.323,Z 1747.495,A 0.000,B 0.000,C 90.000,E1 269.026} C_DIS
LIN {X 0.071,Y -180.888,Z 1747.473,A 0.000,B 0.000,C 90.000,E1 265.122} C_DIS
LIN {X -0.048,Y -179.012,Z 1747.445,A 0.000,B 0.000,C 90.000,E1 260.095} C_DIS
LIN {X 0.048,Y -178.630,Z 1747.440,A 0.000,B 0.000,C 90.000,E1 259.218} C_DIS
LIN {X -0.054,Y -175.681,Z 1747.412,A 0.000,B 0.000,C 90.000,E1 254.157} C_DIS
LIN {X -0.043,Y -172.398,Z 1747.388,A 0.000,B 0.000,C 90.000,E1 249.880} C_DIS
LIN {X -0.026,Y -171.206,Z 1747.379,A 0.000,B 0.000,C 90.000,E1 248.156} C_DIS
LIN {X 0.024,Y -167.493,Z 1747.355,A 0.000,B 0.000,C 90.000,E1 243.819} C_DIS
LIN {X 0.032,Y -166.889,Z 1747.350,A 0.000,B 0.000,C 90.000,E1 242.948} C_DIS
LIN {X 0.023,Y -162.195,Z 1747.321,A 0.000,B 0.000,C 90.000,E1 237.709} C_DIS
LIN {X -0.010,Y -160.767,Z 1747.311,A 0.000,B 0.000,C 90.000,E1 235.960} C_DIS
LIN {X 0.058,Y -157.562,Z 1747.291,A 0.000,B 0.000,C 90.000,E1 232.396} C_DIS
LIN {X -0.004,Y -155.592,Z 1747.276,A 0.000,B 0.000,C 90.000,E1 229.747} C_DIS
LIN {X 0.048,Y -151.875,Z 1747.251,A 0.000,B 0.000,C 90.000,E1 225.243} C_DIS
LIN {X 0.061,Y -150.100,Z 1747.236,A 0.000,B 0.000,C 90.000,E1 222.528} C_DIS
LIN {X -0.022,Y -146.898,Z 1747.211,A 0.000,B 0.000,C 90.000,E1 218.016} C_DIS
LIN {X 0.082,Y -145.485,Z 1747.196,A 0.000,B 0.000,C 90.000,E1 215.231} C_DIS
LIN {X -0.001,Y -142.893,Z 1747.170,A 0.000,B 0.000,C 90.000,E1 210.669} C_DIS
LIN {X -0.071,Y -141.513,Z 1747.150,A 0.000,B 0.000,C 90.000,E1 207.001} C_DIS
LIN {X -0.027,Y -139.393,Z 1747.114,A 0.000,B 0.000,C 90.000,E1 200.482} C_DIS
LIN {X 0.024,Y -139.102,Z 1747.103,A 0.000,B 0.000,C 90.000,E1 198.598} C_DIS
LIN {X 0.016,Y -138.353,Z 1747.057,A 0.000,B 0.000,C 90.000,E1 190.197} C_DIS
LIN {X 0.009,Y -139.513,Z 1747.005,A 0.000,B 0.000,C 90.000,E1 180.859} C_DIS
LIN {X -0.051,Y -141.162,Z 1746.974,A 0.000,B 0.000,C 90.000,E1 175.298} C_DIS
LIN {X 0.062,Y -142.541,Z 1746.958,A 0.000,B 0.000,C 90.000,E1 172.470} C_DIS
LIN {X -0.012,Y -144.814,Z 1746.933,A 0.000,B 0.000,C 90.000,E1 167.881} C_DIS
LIN {X -0.025,Y -147.434,Z 1746.912,A 0.000,B 0.000,C 90.000,E1 164.212} C_DIS
LIN {X 0.003,Y -150.013,Z 1746.892,A 0.000,B 0.000,C 90.000,E1 160.550} C_DIS
LIN {X 0.010,Y -153.346,Z 1746.872,A 0.000,B 0.000,C 90.000,E1 156.922} C_DIS
LIN {X -0.009,Y -155.881,Z 1746.857,A 0.000,B 0.000,C 90.000,E1 154.229} C_DIS
LIN {X -0.042,Y -159.737,Z 1746.837,A 0.000,B 0.000,C 90.000,E1 150.667} C_DIS
LIN {X 0.024,Y -161.976,Z 1746.827,A 0.000,B 0.000,C 90.000,E1 148.869} C_DIS
LIN {X -0.093,Y -166.168,Z 1746.807,A 0.000,B 0.000,C 90.000,E1 145.388} C_DIS
LIN {X -0.098,Y -171.182,Z 1746.788,A 0.000,B 0.000,C 90.000,E1 141.904} C_DIS
LIN {X 0.068,Y -176.063,Z 1746.769,A 0.000,B 0.000,C 90.000,E1 138.405} C_DIS
LIN {X -0.069,Y -180.321,Z 1746.755,A 0.000,B 0.000,C 90.000,E1 135.891} C_DIS
LIN {X -0.098,Y -185.731,Z 1746.736,A 0.000,B 0.000,C 90.000,E1 132.528} C_DIS
LIN {X -0.047,Y -190.340,Z 1746.722,A 0.000,B 0.000,C 90.000,E1 130.011} C_DIS
LIN {X 0.000,Y -197.666,Z 1746.699,A 0.000,B 0.000,C 90.000,E1 125.884} C_DIS
LIN {X 0.042,Y -200.920,Z 1746.690,A 0.000,B 0.000,C 90.000,E1 124.246} C_DIS
LIN {X -0.047,Y -206.825,Z 1746.672,A 0.000,B 0.000,C 90.000,E1 121.052} C_DIS
LIN {X -0.039,Y -210.355,Z 1746.663,A 0.000,B 0.000,C 90.000,E1 119.333} C_DIS
LIN {X -0.098,Y -334.953,Z 1746.663,A 0.000,B 0.000,C 90.000,E1 119.333} C_DIS
LIN {X -0.070,Y -338.082,Z 1746.663,A 0.000,B 0.000,C 90.000,E1 119.283} C_DIS
LIN {X 0.077,Y -343.810,Z 1746.661,A 0.000,B 0.000,C 90.000,E1 118.949} C_DIS
LIN {X 0.227,Y -346.849,Z 1746.659,A 0.000,B 0.000,C 90.000,E1 118.615} C_DIS
LIN {X 0.099,Y -348.826,Z 1746.658,A 0.000,B 0.000,C 90.000,E1 118.359} C_DIS
LIN {X -0.031,Y -350.369,Z 1746.656,A 0.000,B 0.000,C 90.000,E1 118.103} C_DIS
LIN {X -0.173,Y -363.435,Z 1746.641,A 0.000,B 0.000,C 90.000,E1 115.412} C_DIS
LIN {X 0.080,Y -378.011,Z 1746.626,A 0.000,B 0.000,C 90.000,E1 112.717} C_DIS
LIN {X -0.049,Y -392.355,Z 1746.613,A 0.000,B 0.000,C 90.000,E1 110.429} C_DIS
LIN {X -0.108,Y -408.107,Z 1746.601,A 0.000,B 0.000,C 90.000,E1 108.181} C_DIS
LIN {X -0.027,Y -425.375,Z 1746.589,A 0.000,B 0.000,C 90.000,E1 105.969} C_DIS
LIN {X -0.049,Y -444.280,Z 1746.577,A 0.000,B 0.000,C 90.000,E1 103.828} C_DIS
LIN {X -0.182,Y -464.243,Z 1746.566,A 0.000,B 0.000,C 90.000,E1 101.827} C_DIS
LIN {X 0.029,Y -487.336,Z 1746.554,A 0.000,B 0.000,C 90.000,E1 99.726} C_DIS
LIN {X 0.196,Y -510.888,Z 1746.544,A 0.000,B 0.000,C 90.000,E1 97.814} C_DIS
LIN {X 0.060,Y -514.384,Z 1746.541,A 0.000,B 0.000,C 90.000,E1 97.409} C_DIS
LIN {X -0.051,Y -515.705,Z 1746.540,A 0.000,B 0.000,C 90.000,E1 97.182} C_DIS
LIN {X -0.097,Y -516.671,Z 1746.539,A 0.000,B 0.000,C 90.000,E1 96.947} C_DIS
LIN {X -0.228,Y -517.719,Z 1746.536,A 0.000,B 0.000,C 90.000,E1 96.486} C_DIS
LIN {X 0.159,Y -517.725,Z 1746.533,A 0.000,B 0.000,C 90.000,E1 95.967} C_DIS
LIN {X -0.012,Y -516.689,Z 1746.531,A 0.000,B 0.000,C 90.000,E1 95.511} C_DIS
LIN {X -0.048,Y -515.730,Z 1746.529,A 0.000,B 0.000,C 90.000,E1 95.277} C_DIS
LIN {X -0.130,Y -514.413,Z 1746.528,A 0.000,B 0.000,C 90.000,E1 95.049} C_DIS
LIN {X -0.108,Y -503.645,Z 1746.520,A 0.000,B 0.000,C 90.000,E1 93.612} C_DIS
LIN {X 0.204,Y -492.927,Z 1746.512,A 0.000,B 0.000,C 90.000,E1 92.121} C_DIS
LIN {X 0.161,Y -480.078,Z 1746.502,A 0.000,B 0.000,C 90.000,E1 90.401} C_DIS
LIN {X -0.133,Y -467.313,Z 1746.493,A 0.000,B 0.000,C 90.000,E1 88.682} C_DIS
LIN {X -0.205,Y -454.457,Z 1746.483,A 0.000,B 0.000,C 90.000,E1 86.906} C_DIS
LIN {X -0.021,Y -441.637,Z 1746.473,A 0.000,B 0.000,C 90.000,E1 85.065} C_DIS
LIN {X 0.085,Y -427.145,Z 1746.461,A 0.000,B 0.000,C 90.000,E1 82.932} C_DIS
LIN {X -0.094,Y -413.004,Z 1746.449,A 0.000,B 0.000,C 90.000,E1 80.792} C_DIS
LIN {X 0.187,Y -394.567,Z 1746.432,A 0.000,B 0.000,C 90.000,E1 77.701} C_DIS
LIN {X 0.102,Y -378.760,Z 1746.416,A 0.000,B 0.000,C 90.000,E1 74.866} C_DIS
LIN {X 0.055,Y -366.494,Z 1746.403,A 0.000,B 0.000,C 90.000,E1 72.543} C_DIS
LIN {X -0.066,Y -354.569,Z 1746.390,A 0.000,B 0.000,C 90.000,E1 70.188} C_DIS
LIN {X -0.058,Y -339.016,Z 1746.371,A 0.000,B 0.000,C 90.000,E1 66.847} C_DIS
LIN {X 0.117,Y -328.051,Z 1746.358,A 0.000,B 0.000,C 90.000,E1 64.332} C_DIS
LIN {X 0.010,Y -317.230,Z 1746.344,A 0.000,B 0.000,C 90.000,E1 61.820} C_DIS
LIN {X 0.050,Y -310.416,Z 1746.334,A 0.000,B 0.000,C 90.000,E1 60.205} C_DIS
LIN {X 0.091,Y -300.416,Z 1746.322,A 0.000,B 0.000,C 90.000,E1 57.916} C_DIS
LIN {X 0.065,Y -289.004,Z 1746.307,A 0.000,B 0.000,C 90.000,E1 55.261} C_DIS
LIN {X -0.110,Y -278.985,Z 1746.294,A 0.000,B 0.000,C 90.000,E1 52.924} C_DIS
LIN {X 0.137,Y -270.655,Z 1746.282,A 0.000,B 0.000,C 90.000,E1 50.803} C_DIS
LIN {X -0.038,Y -258.409,Z 1746.265,A 0.000,B 0.000,C 90.000,E1 47.676} C_DIS
LIN {X -0.028,Y -247.885,Z 1746.249,A 0.000,B 0.000,C 90.000,E1 44.798} C_DIS
LIN {X 0.044,Y -236.544,Z 1746.230,A 0.000,B 0.000,C 90.000,E1 41.472} C_DIS
LIN {X 0.012,Y -225.884,Z 1746.212,A 0.000,B 0.000,C 90.000,E1 38.096} C_DIS
LIN {X 0.022,Y -217.092,Z 1746.195,A 0.000,B 0.000,C 90.000,E1 35.025} C_DIS
LIN {X -0.056,Y -209.125,Z 1746.177,A 0.000,B 0.000,C 90.000,E1 31.926} C_DIS
LIN {X -0.016,Y -201.955,Z 1746.160,A 0.000,B 0.000,C 90.000,E1 28.743} C_DIS
LIN {X -0.079,Y -195.436,Z 1746.142,A 0.000,B 0.000,C 90.000,E1 25.540} C_DIS
LIN {X -0.034,Y -189.664,Z 1746.124,A 0.000,B 0.000,C 90.000,E1 22.259} C_DIS
LIN {X -0.070,Y -184.695,Z 1746.105,A 0.000,B 0.000,C 90.000,E1 18.960} C_DIS
LIN {X -0.048,Y -180.449,Z 1746.087,A 0.000,B 0.000,C 90.000,E1 15.607} C_DIS
LIN {X -0.093,Y -177.091,Z 1746.068,A 0.000,B 0.000,C 90.000,E1 12.243} C_DIS
LIN {X 0.056,Y -173.886,Z 1746.044,A 0.000,B 0.000,C 90.000,E1 7.936} C_DIS
LIN {X -0.011,Y -171.291,Z 1746.016,A 0.000,B 0.000,C 90.000,E1 2.808} C_DIS
LIN {X -0.086,Y -170.163,Z 1745.973,A 0.000,B 0.000,C 90.000,E1 355.241} C_DIS
LIN {X 0.083,Y -171.289,Z 1745.930,A 0.000,B 0.000,C 90.000,E1 347.409} C_DIS
LIN {X 0.028,Y -173.842,Z 1745.897,A 0.000,B 0.000,C 90.000,E1 341.402} C_DIS
LIN {X 0.094,Y -176.873,Z 1745.873,A 0.000,B 0.000,C 90.000,E1 337.102} C_DIS
LIN {X 0.046,Y -180.731,Z 1745.849,A 0.000,B 0.000,C 90.000,E1 332.871} C_DIS
LIN {X -0.068,Y -184.591,Z 1745.831,A 0.000,B 0.000,C 90.000,E1 329.537} C_DIS
LIN {X 0.033,Y -189.283,Z 1745.812,A 0.000,B 0.000,C 90.000,E1 326.167} C_DIS
LIN {X 0.103,Y -194.932,Z 1745.794,A 0.000,B 0.000,C 90.000,E1 322.844} C_DIS
LIN {X -0.030,Y -201.773,Z 1745.776,A 0.000,B 0.000,C 90.000,E1 319.622} C_DIS
LIN {X 0.075,Y -208.749,Z 1745.760,A 0.000,B 0.000,C 90.000,E1 316.782} C_DIS
LIN {X -0.003,Y -215.541,Z 1745.747,A 0.000,B 0.000,C 90.000,E1 314.433} C_DIS
LIN {X -0.014,Y -222.013,Z 1745.736,A 0.000,B 0.000,C 90.000,E1 312.486} C_DIS
LIN {X 0.086,Y -229.353,Z 1745.725,A 0.000,B 0.000,C 90.000,E1 310.539} C_DIS
LIN {X -0.008,Y -237.738,Z 1745.715,A 0.000,B 0.000,C 90.000,E1 308.669} C_DIS
LIN {X -0.080,Y -249.143,Z 1745.702,A 0.000,B 0.000,C 90.000,E1 306.457} C_DIS
LIN {X -0.075,Y -261.728,Z 1745.690,A 0.000,B 0.000,C 90.000,E1 304.278} C_DIS
LIN {X -0.041,Y -277.641,Z 1745.677,A 0.000,B 0.000,C 90.000,E1 301.799} C_DIS
LIN {X -0.104,Y -297.273,Z 1745.661,A 0.000,B 0.000,C 90.000,E1 299.077} C_DIS
LIN {X 0.000,Y -315.413,Z 1745.649,A 0.000,B 0.000,C 90.000,E1 296.744} C_DIS
LIN {X 0.004,Y -331.391,Z 1745.638,A 0.000,B 0.000,C 90.000,E1 294.823} C_DIS
LIN {X 0.054,Y -344.470,Z 1745.629,A 0.000,B 0.000,C 90.000,E1 293.259} C_DIS
LIN {X 0.164,Y -354.724,Z 1745.623,A 0.000,B 0.000,C 90.000,E1 292.025} C_DIS
LIN {X 0.016,Y -364.634,Z 1745.616,A 0.000,B 0.000,C 90.000,E1 290.844} C_DIS
LIN {X 0.107,Y -371.689,Z 1745.611,A 0.000,B 0.000,C 90.000,E1 289.939} C_DIS
LIN {X -0.077,Y -378.080,Z 1745.606,A 0.000,B 0.000,C 90.000,E1 289.087} C_DIS
LIN {X 0.150,Y -383.670,Z 1745.601,A 0.000,B 0.000,C 90.000,E1 288.181} C_DIS
LIN {X -0.071,Y -386.851,Z 1745.598,A 0.000,B 0.000,C 90.000,E1 287.638} C_DIS
LIN {X 0.097,Y -389.564,Z 1745.595,A 0.000,B 0.000,C 90.000,E1 287.040} C_DIS
LIN {X -0.092,Y -391.837,Z 1745.592,A 0.000,B 0.000,C 90.000,E1 286.496} C_DIS
LIN {X 0.111,Y -393.728,Z 1745.588,A 0.000,B 0.000,C 90.000,E1 285.898} C_DIS
LIN {X -0.166,Y -395.284,Z 1745.585,A 0.000,B 0.000,C 90.000,E1 285.371} C_DIS
LIN {X 0.055,Y -396.507,Z 1745.582,A 0.000,B 0.000,C 90.000,E1 284.773} C_DIS
LIN {X -0.199,Y -397.376,Z 1745.579,A 0.000,B 0.000,C 90.000,E1 284.245} C_DIS
LIN {X 0.037,Y -397.892,Z 1745.576,A 0.000,B 0.000,C 90.000,E1 283.647} C_DIS
LIN {X 0.183,Y -398.047,Z 1745.573,A 0.000,B 0.000,C 90.000,E1 283.063} C_DIS
LIN {X -0.053,Y -397.763,Z 1745.570,A 0.000,B 0.000,C 90.000,E1 282.535} C_DIS
LIN {X 0.101,Y -397.039,Z 1745.567,A 0.000,B 0.000,C 90.000,E1 281.951} C_DIS
LIN {X -0.136,Y -395.842,Z 1745.563,A 0.000,B 0.000,C 90.000,E1 281.422} C_DIS
LIN {X 0.012,Y -394.145,Z 1745.560,A 0.000,B 0.000,C 90.000,E1 280.838} C_DIS
LIN {X 0.149,Y -391.814,Z 1745.557,A 0.000,B 0.000,C 90.000,E1 280.254} C_DIS
LIN {X -0.116,Y -388.836,Z 1745.554,A 0.000,B 0.000,C 90.000,E1 279.726} C_DIS
LIN {X 0.004,Y -382.137,Z 1745.548,A 0.000,B 0.000,C 90.000,E1 278.568} C_DIS
LIN {X 0.044,Y -376.336,Z 1745.541,A 0.000,B 0.000,C 90.000,E1 277.409} C_DIS
LIN {X 0.013,Y -372.896,Z 1745.538,A 0.000,B 0.000,C 90.000,E1 276.834} C_DIS
LIN {X -0.034,Y -368.837,Z 1745.535,A 0.000,B 0.000,C 90.000,E1 276.258} C_DIS
LIN {X -0.102,Y -363.932,Z 1745.531,A 0.000,B 0.000,C 90.000,E1 275.682} C_DIS
LIN {X 0.162,Y -358.338,Z 1745.528,A 0.000,B 0.000,C 90.000,E1 275.049} C_DIS
LIN {X -0.032,Y -352.452,Z 1745.525,A 0.000,B 0.000,C 90.000,E1 274.531} C_DIS
LIN {X -0.027,Y -343.433,Z 1745.521,A 0.000,B 0.000,C 90.000,E1 273.784} C_DIS
LIN {X -0.019,Y -337.340,Z 1745.518,A 0.000,B 0.000,C 90.000,E1 273.326} C_DIS
LIN {X -0.134,Y -330.992,Z 1745.516,A 0.000,B 0.000,C 90.000,E1 272.922} C_DIS
LIN {X -0.063,Y -324.481,Z 1745.514,A 0.000,B 0.000,C 90.000,E1 272.522} C_DIS
LIN {X -0.102,Y -317.740,Z 1745.512,A 0.000,B 0.000,C 90.000,E1 272.178} C_DIS
LIN {X 0.113,Y -310.707,Z 1745.510,A 0.000,B 0.000,C 90.000,E1 271.835} C_DIS
LIN {X -0.046,Y -303.550,Z 1745.509,A 0.000,B 0.000,C 90.000,E1 271.604} C_DIS
LIN {X 0.090,Y -292.607,Z 1745.507,A 0.000,B 0.000,C 90.000,E1 271.260} C_DIS
LIN {X 0.011,Y -281.270,Z 1745.506,A 0.000,B 0.000,C 90.000,E1 271.031} C_DIS
LIN {X -0.092,Y -272.741,Z 1745.505,A 0.000,B 0.000,C 90.000,E1 270.917} C_DIS
LIN {X -0.032,Y -252.415,Z 1745.504,A 0.000,B 0.000,C 90.000,E1 270.688} C_DIS
LIN {X 0.050,Y -237.885,Z 1745.503,A 0.000,B 0.000,C 90.000,E1 270.573} C_DIS
LIN {X 0.027,Y -235.432,Z 1745.503,A 0.000,B 0.000,C 90.000,E1 270.573} C_DIS
LIN {X 0.002,Y -181.553,Z 1745.503,A 0.000,B 0.000,C 90.000,E1 270.573} C_DIS
LIN {X 0.005,Y -181.287,Z 1745.494,A 0.000,B 0.000,C 90.000,E1 268.854} C_DIS
LIN {X 0.053,Y -180.907,Z 1745.475,A 0.000,B 0.000,C 90.000,E1 265.469} C_DIS
LIN {X -0.070,Y -180.744,Z 1745.470,A 0.000,B 0.000,C 90.000,E1 264.666} C_DIS
LIN {X 0.031,Y -178.835,Z 1745.442,A 0.000,B 0.000,C 90.000,E1 259.567} C_DIS
LIN {X -0.105,Y -175.879,Z 1745.414,A 0.000,B 0.000,C 90.000,E1 254.519} C_DIS
LIN {X 0.002,Y -174.541,Z 1745.404,A 0.000,B 0.000,C 90.000,E1 252.779} C_DIS
LIN {X 0.094,Y -171.525,Z 1745.380,A 0.000,B 0.000,C 90.000,E1 248.465} C_DIS
LIN {X 0.080,Y -167.751,Z 1745.357,A 0.000,B 0.000,C 90.000,E1 244.152} C_DIS
LIN {X 0.018,Y -166.454,Z 1745.347,A 0.000,B 0.000,C 90.000,E1 242.436} C_DIS
LIN {X 0.008,Y -163.170,Z 1745.328,A 0.000,B 0.000,C 90.000,E1 238.948} C_DIS
LIN {X 0.058,Y -161.129,Z 1745.313,A 0.000,B 0.000,C 90.000,E1 236.294} C_DIS
LIN {X -0.040,Y -157.151,Z 1745.288,A 0.000,B 0.000,C 90.000,E1 231.904} C_DIS
LIN {X -0.017,Y -155.883,Z 1745.278,A 0.000,B 0.000,C 90.000,E1 230.114} C_DIS
LIN {X -0.058,Y -152.133,Z 1745.254,A 0.000,B 0.000,C 90.000,E1 225.648} C_DIS
LIN {X -0.038,Y -150.383,Z 1745.238,A 0.000,B 0.000,C 90.000,E1 222.933} C_DIS
LIN {X -0.013,Y -147.116,Z 1745.213,A 0.000,B 0.000,C 90.000,E1 218.382} C_DIS
LIN {X -0.023,Y -145.681,Z 1745.198,A 0.000,B 0.000,C 90.000,E1 215.644} C_DIS
LIN {X -0.024,Y -143.063,Z 1745.172,A 0.000,B 0.000,C 90.000,E1 211.052} C_DIS
LIN {X 0.033,Y -141.684,Z 1745.152,A 0.000,B 0.000,C 90.000,E1 207.334} C_DIS
LIN {X 0.011,Y -139.458,Z 1745.116,A 0.000,B 0.000,C 90.000,E1 200.844} C_DIS
LIN {X 0.062,Y -139.192,Z 1745.105,A 0.000,B 0.000,C 90.000,E1 198.960} C_DIS
LIN {X -0.051,Y -138.325,Z 1745.054,A 0.000,B 0.000,C 90.000,E1 189.670} C_DIS
LIN {X -0.046,Y -139.454,Z 1745.007,A 0.000,B 0.000,C 90.000,E1 181.260} C_DIS
LIN {X 0.033,Y -141.001,Z 1744.976,A 0.000,B 0.000,C 90.000,E1 175.641} C_DIS
LIN {X -0.016,Y -142.756,Z 1744.955,A 0.000,B 0.000,C 90.000,E1 171.951} C_DIS
LIN {X -0.060,Y -145.158,Z 1744.930,A 0.000,B 0.000,C 90.000,E1 167.353} C_DIS
LIN {X -0.068,Y -147.781,Z 1744.909,A 0.000,B 0.000,C 90.000,E1 163.685} C_DIS
LIN {X 0.011,Y -150.459,Z 1744.889,A 0.000,B 0.000,C 90.000,E1 160.007} C_DIS
LIN {X 0.085,Y -153.909,Z 1744.869,A 0.000,B 0.000,C 90.000,E1 156.357} C_DIS
LIN {X 0.010,Y -157.320,Z 1744.849,A 0.000,B 0.000,C 90.000,E1 152.794} C_DIS
LIN {X -0.044,Y -161.508,Z 1744.829,A 0.000,B 0.000,C 90.000,E1 149.253} C_DIS
LIN {X -0.028,Y -165.707,Z 1744.810,A 0.000,B 0.000,C 90.000,E1 145.722} C_DIS
LIN {X 0.097,Y -170.653,Z 1744.790,A 0.000,B 0.000,C 90.000,E1 142.190} C_DIS
LIN {X 0.010,Y -175.528,Z 1744.771,A 0.000,B 0.000,C 90.000,E1 138.771} C_DIS
LIN {X 0.004,Y -181.148,Z 1744.752,A 0.000,B 0.000,C 90.000,E1 135.364} C_DIS
LIN {X 0.001,Y -186.600,Z 1744.733,A 0.000,B 0.000,C 90.000,E1 132.000} C_DIS
LIN {X 0.071,Y -191.211,Z 1744.719,A 0.000,B 0.000,C 90.000,E1 129.483} C_DIS
LIN {X -0.005,Y -197.023,Z 1744.701,A 0.000,B 0.000,C 90.000,E1 126.217} C_DIS
LIN {X -0.087,Y -200.294,Z 1744.692,A 0.000,B 0.000,C 90.000,E1 124.612} C_DIS
LIN {X -0.094,Y -207.785,Z 1744.670,A 0.000,B 0.000,C 90.000,E1 120.590} C_DIS
LIN {X 0.044,Y -210.314,Z 1744.663,A 0.000,B 0.000,C 90.000,E1 119.333} C_DIS
LIN {X 0.016,Y -335.959,Z 1744.663,A 0.000,B 0.000,C 90.000,E1 119.333} C_DIS
LIN {X -0.145,Y -337.525,Z 1744.663,A 0.000,B 0.000,C 90.000,E1 119.333} C_DIS
LIN {X -0.082,Y -341.525,Z 1744.662,A 0.000,B 0.000,C 90.000,E1 119.155} C_DIS
LIN {X 0.150,Y -343.842,Z 1744.661,A 0.000,B 0.000,C 90.000,E1 118.949} C_DIS
LIN {X -0.089,Y -347.694,Z 1744.659,A 0.000,B 0.000,C 90.000,E1 118.565} C_DIS
LIN {X 0.157,Y -349.536,Z 1744.657,A 0.000,B 0.000,C 90.000,E1 118.231} C_DIS
LIN {X 0.023,Y -365.641,Z 1744.639,A 0.000,B 0.000,C 90.000,E1 114.951} C_DIS
LIN {X -0.157,Y -380.470,Z 1744.624,A 0.000,B 0.000,C 90.000,E1 112.333} C_DIS
LIN {X 0.129,Y -395.059,Z 1744.611,A 0.000,B 0.000,C 90.000,E1 109.993} C_DIS
LIN {X 0.010,Y -411.075,Z 1744.599,A 0.000,B 0.000,C 90.000,E1 107.764} C_DIS
LIN {X -0.238,Y -428.628,Z 1744.587,A 0.000,B 0.000,C 90.000,E1 105.607} C_DIS
LIN {X -0.161,Y -447.797,Z 1744.575,A 0.000,B 0.000,C 90.000,E1 103.467} C_DIS
LIN {X -0.159,Y -467.863,Z 1744.564,A 0.000,B 0.000,C 90.000,E1 101.478} C_DIS
LIN {X -0.184,Y -491.086,Z 1744.552,A 0.000,B 0.000,C 90.000,E1 99.434} C_DIS
LIN {X 0.119,Y -509.522,Z 1744.544,A 0.000,B 0.000,C 90.000,E1 97.936} C_DIS
LIN {X -0.093,Y -511.696,Z 1744.543,A 0.000,B 0.000,C 90.000,E1 97.757} C_DIS
LIN {X -0.108,Y -513.555,Z 1744.542,A 0.000,B 0.000,C 90.000,E1 97.530} C_DIS
LIN {X -0.055,Y -514.962,Z 1744.541,A 0.000,B 0.000,C 90.000,E1 97.296} C_DIS
LIN {X -0.197,Y -516.838,Z 1744.538,A 0.000,B 0.000,C 90.000,E1 96.834} C_DIS
LIN {X 0.183,Y -517.566,Z 1744.535,A 0.000,B 0.000,C 90.000,E1 96.315} C_DIS
LIN {X 0.058,Y -517.271,Z 1744.533,A 0.000,B 0.000,C 90.000,E1 95.853} C_DIS
LIN {X -0.064,Y -515.897,Z 1744.530,A 0.000,B 0.000,C 90.000,E1 95.391} C_DIS
LIN {X -0.149,Y -514.734,Z 1744.529,A 0.000,B 0.000,C 90.000,E1 95.163} C_DIS
LIN {X 0.231,Y -511.364,Z 1744.526,A 0.000,B 0.000,C 90.000,E1 94.645} C_DIS
LIN {X -0.168,Y -495.182,Z 1744.514,A 0.000,B 0.000,C 90.000,E1 92.522} C_DIS
LIN {X -0.002,Y -484.251,Z 1744.506,A 0.000,B 0.000,C 90.000,E1 91.031} C_DIS
LIN {X 0.070,Y -469.622,Z 1744.495,A 0.000,B 0.000,C 90.000,E1 89.026} C_DIS
LIN {X 0.041,Y -456.765,Z 1744.485,A 0.000,B 0.000,C 90.000,E1 87.249} C_DIS
LIN {X 0.011,Y -442.122,Z 1744.473,A 0.000,B 0.000,C 90.000,E1 85.179} C_DIS
LIN {X 0.077,Y -427.590,Z 1744.461,A 0.000,B 0.000,C 90.000,E1 83.053} C_DIS
LIN {X -0.037,Y -413.408,Z 1744.449,A 0.000,B 0.000,C 90.000,E1 80.905} C_DIS
LIN {X -0.202,Y -394.922,Z 1744.432,A 0.000,B 0.000,C 90.000,E1 77.881} C_DIS
LIN {X 0.099,Y -379.078,Z 1744.417,A 0.000,B 0.000,C 90.000,E1 74.991} C_DIS
LIN {X 0.054,Y -366.773,Z 1744.404,A 0.000,B 0.000,C 90.000,E1 72.670} C_DIS
LIN {X 0.054,Y -354.815,Z 1744.391,A 0.000,B 0.000,C 90.000,E1 70.296} C_DIS
LIN {X -0.058,Y -339.211,Z 1744.372,A 0.000,B 0.000,C 90.000,E1 66.975} C_DIS
LIN {X 0.010,Y -329.574,Z 1744.360,A 0.000,B 0.000,C 90.000,E1 64.793} C_DIS
LIN {X -0.065,Y -318.692,Z 1744.346,A 0.000,B 0.000,C 90.000,E1 62.281} C_DIS
LIN {X 0.063,Y -310.550,Z 1744.335,A 0.000,B 0.000,C 90.000,E1 60.333} C_DIS
LIN {X -0.082,Y -302.016,Z 1744.324,A 0.000,B 0.000,C 90.000,E1 58.408} C_DIS
LIN {X -0.065,Y -292.059,Z 1744.312,A 0.000,B 0.000,C 90.000,E1 56.087} C_DIS
LIN {X -0.069,Y -283.497,Z 1744.300,A 0.000,B 0.000,C 90.000,E1 54.069} C_DIS
LIN {X -0.087,Y -272.296,Z 1744.285,A 0.000,B 0.000,C 90.000,E1 51.331} C_DIS
LIN {X -0.075,Y -261.263,Z 1744.270,A 0.000,B 0.000,C 90.000,E1 48.528} C_DIS
LIN {X 0.175,Y -251.965,Z 1744.256,A 0.000,B 0.000,C 90.000,E1 45.972} C_DIS
LIN {X 0.017,Y -241.622,Z 1744.239,A 0.000,B 0.000,C 90.000,E1 43.095} C_DIS
LIN {X 0.097,Y -230.628,Z 1744.221,A 0.000,B 0.000,C 90.000,E1 39.725} C_DIS
LIN {X 0.108,Y -220.359,Z 1744.202,A 0.000,B 0.000,C 90.000,E1 36.297} C_DIS
LIN {X 0.042,Y -212.100,Z 1744.185,A 0.000,B 0.000,C 90.000,E1 33.214} C_DIS
LIN {X -0.024,Y -204.629,Z 1744.167,A 0.000,B 0.000,C 90.000,E1 30.079} C_DIS
LIN {X -0.012,Y -197.874,Z 1744.149,A 0.000,B 0.000,C 90.000,E1 26.873} C_DIS
LIN {X -0.081,Y -191.810,Z 1744.131,A 0.000,B 0.000,C 90.000,E1 23.643} C_DIS
LIN {X 0.074,Y -186.502,Z 1744.113,A 0.000,B 0.000,C 90.000,E1 20.301} C_DIS
LIN {X 0.019,Y -181.955,Z 1744.094,A 0.000,B 0.000,C 90.000,E1 16.985} C_DIS
LIN {X -0.075,Y -178.244,Z 1744.076,A 0.000,B 0.000,C 90.000,E1 13.647} C_DIS
LIN {X -0.008,Y -174.687,Z 1744.052,A 0.000,B 0.000,C 90.000,E1 9.378} C_DIS
LIN {X -0.033,Y -171.679,Z 1744.024,A 0.000,B 0.000,C 90.000,E1 4.245} C_DIS
LIN {X -0.091,Y -169.967,Z 1743.973,A 0.000,B 0.000,C 90.000,E1 355.241} C_DIS
LIN {X -0.062,Y -171.365,Z 1743.925,A 0.000,B 0.000,C 90.000,E1 346.589} C_DIS
LIN {X -0.016,Y -174.215,Z 1743.892,A 0.000,B 0.000,C 90.000,E1 340.550} C_DIS
LIN {X -0.036,Y -177.436,Z 1743.868,A 0.000,B 0.000,C 90.000,E1 336.282} C_DIS
LIN {X 0.014,Y -181.493,Z 1743.845,A 0.000,B 0.000,C 90.000,E1 332.025} C_DIS
LIN {X 0.011,Y -185.582,Z 1743.826,A 0.000,B 0.000,C 90.000,E1 328.663} C_DIS
LIN {X 0.087,Y -190.578,Z 1743.807,A 0.000,B 0.000,C 90.000,E1 325.308} C_DIS
LIN {X 0.059,Y -194.930,Z 1743.794,A 0.000,B 0.000,C 90.000,E1 322.844} C_DIS
LIN {X -0.076,Y -201.843,Z 1743.776,A 0.000,B 0.000,C 90.000,E1 319.622} C_DIS
LIN {X 0.062,Y -209.956,Z 1743.758,A 0.000,B 0.000,C 90.000,E1 316.377} C_DIS
LIN {X 0.008,Y -216.952,Z 1743.745,A 0.000,B 0.000,C 90.000,E1 314.028} C_DIS
LIN {X 0.023,Y -223.620,Z 1743.734,A 0.000,B 0.000,C 90.000,E1 312.081} C_DIS
LIN {X -0.008,Y -231.195,Z 1743.723,A 0.000,B 0.000,C 90.000,E1 310.172} C_DIS
LIN {X -0.069,Y -239.788,Z 1743.713,A 0.000,B 0.000,C 90.000,E1 308.302} C_DIS
LIN {X 0.039,Y -249.397,Z 1743.702,A 0.000,B 0.000,C 90.000,E1 306.423} C_DIS
LIN {X 0.046,Y -261.945,Z 1743.690,A 0.000,B 0.000,C 90.000,E1 304.246} C_DIS
LIN {X -0.131,Y -280.228,Z 1743.675,A 0.000,B 0.000,C 90.000,E1 301.465} C_DIS
LIN {X 0.131,Y -300.060,Z 1743.660,A 0.000,B 0.000,C 90.000,E1 298.693} C_DIS
LIN {X -0.047,Y -320.993,Z 1743.645,A 0.000,B 0.000,C 90.000,E1 296.104} C_DIS
LIN {X -0.034,Y -334.230,Z 1743.636,A 0.000,B 0.000,C 90.000,E1 294.515} C_DIS
LIN {X 0.040,Y -347.334,Z 1743.628,A 0.000,B 0.000,C 90.000,E1 292.950} C_DIS
LIN {X 0.141,Y -357.528,Z 1743.621,A 0.000,B 0.000,C 90.000,E1 291.716} C_DIS
LIN {X -0.035,Y -367.211,Z 1743.614,A 0.000,B 0.000,C 90.000,E1 290.556} C_DIS
LIN {X -0.133,Y -374.142,Z 1743.609,A 0.000,B 0.000,C 90.000,E1 289.685} C_DIS
LIN {X 0.051,Y -380.279,Z 1743.604,A 0.000,B 0.000,C 90.000,E1 288.779} C_DIS
LIN {X 0.172,Y -383.923,Z 1743.601,A 0.000,B 0.000,C 90.000,E1 288.181} C_DIS
LIN {X -0.048,Y -387.107,Z 1743.598,A 0.000,B 0.000,C 90.000,E1 287.638} C_DIS
LIN {X 0.123,Y -389.817,Z 1743.595,A 0.000,B 0.000,C 90.000,E1 287.040} C_DIS
LIN {X -0.064,Y -392.105,Z 1743.592,A 0.000,B 0.000,C 90.000,E1 286.496} C_DIS
LIN {X 0.141,Y -394.002,Z 1743.588,A 0.000,B 0.000,C 90.000,E1 285.898} C_DIS
LIN {X -0.135,Y -395.540,Z 1743.585,A 0.000,B 0.000,C 90.000,E1 285.371} C_DIS
LIN {X 0.088,Y -396.799,Z 1743.582,A 0.000,B 0.000,C 90.000,E1 284.773} C_DIS
LIN {X -0.165,Y -397.650,Z 1743.579,A 0.000,B 0.000,C 90.000,E1 284.245} C_DIS
LIN {X 0.073,Y -398.159,Z 1743.576,A 0.000,B 0.000,C 90.000,E1 283.647} C_DIS
LIN {X -0.167,Y -398.319,Z 1743.573,A 0.000,B 0.000,C 90.000,E1 283.119} C_DIS
LIN {X -0.013,Y -398.058,Z 1743.570,A 0.000,B 0.000,C 90.000,E1 282.535} C_DIS
LIN {X 0.142,Y -397.329,Z 1743.567,A 0.000,B 0.000,C 90.000,E1 281.951} C_DIS
LIN {X -0.093,Y -396.130,Z 1743.563,A 0.000,B 0.000,C 90.000,E1 281.422} C_DIS
LIN {X 0.056,Y -394.415,Z 1743.560,A 0.000,B 0.000,C 90.000,E1 280.838} C_DIS
LIN {X 0.195,Y -392.106,Z 1743.557,A 0.000,B 0.000,C 90.000,E1 280.254} C_DIS
LIN {X -0.069,Y -389.131,Z 1743.554,A 0.000,B 0.000,C 90.000,E1 279.726} C_DIS
LIN {X 0.054,Y -382.421,Z 1743.548,A 0.000,B 0.000,C 90.000,E1 278.568} C_DIS
LIN {X 0.095,Y -376.533,Z 1743.541,A 0.000,B 0.000,C 90.000,E1 277.409} C_DIS
LIN {X 0.066,Y -373.080,Z 1743.538,A 0.000,B 0.000,C 90.000,E1 276.834} C_DIS
LIN {X 0.019,Y -368.968,Z 1743.535,A 0.000,B 0.000,C 90.000,E1 276.258} C_DIS
LIN {X -0.049,Y -364.020,Z 1743.531,A 0.000,B 0.000,C 90.000,E1 275.682} C_DIS
LIN {X -0.134,Y -358.440,Z 1743.528,A 0.000,B 0.000,C 90.000,E1 275.106} C_DIS
LIN {X 0.027,Y -352.539,Z 1743.525,A 0.000,B 0.000,C 90.000,E1 274.531} C_DIS
LIN {X 0.042,Y -343.493,Z 1743.521,A 0.000,B 0.000,C 90.000,E1 273.784} C_DIS
LIN {X 0.040,Y -337.391,Z 1743.519,A 0.000,B 0.000,C 90.000,E1 273.326} C_DIS
LIN {X -0.093,Y -330.977,Z 1743.516,A 0.000,B 0.000,C 90.000,E1 272.922} C_DIS
LIN {X -0.024,Y -324.442,Z 1743.514,A 0.000,B 0.000,C 90.000,E1 272.522} C_DIS
LIN {X -0.057,Y -317.629,Z 1743.512,A 0.000,B 0.000,C 90.000,E1 272.178} C_DIS
LIN {X -0.157,Y -310.560,Z 1743.510,A 0.000,B 0.000,C 90.000,E1 271.892} C_DIS
LIN {X -0.018,Y -303.303,Z 1743.509,A 0.000,B 0.000,C 90.000,E1 271.604} C_DIS
LIN {X 0.117,Y -292.178,Z 1743.507,A 0.000,B 0.000,C 90.000,E1 271.260} C_DIS
LIN {X 0.052,Y -280.830,Z 1743.506,A 0.000,B 0.000,C 90.000,E1 271.031} C_DIS
LIN {X -0.039,Y -272.290,Z 1743.505,A 0.000,B 0.000,C 90.000,E1 270.917} C_DIS
LIN {X 0.029,Y -251.981,Z 1743.504,A 0.000,B 0.000,C 90.000,E1 270.688} C_DIS
LIN {X -0.080,Y -239.129,Z 1743.503,A 0.000,B 0.000,C 90.000,E1 270.630} C_DIS
LIN {X 0.109,Y -234.985,Z 1743.503,A 0.000,B 0.000,C 90.000,E1 270.573} C_DIS
LIN {X 0.049,Y -181.551,Z 1743.503,A 0.000,B 0.000,C 90.000,E1 270.573} C_DIS
LIN {X 0.052,Y -181.290,Z 1743.494,A 0.000,B 0.000,C 90.000,E1 268.854} C_DIS
LIN {X -0.079,Y -180.907,Z 1743.475,A 0.000,B 0.000,C 90.000,E1 265.527} C_DIS
LIN {X -0.022,Y -180.751,Z 1743.470,A 0.000,B 0.000,C 90.000,E1 264.666} C_DIS
LIN {X 0.047,Y -178.842,Z 1743.442,A 0.000,B 0.000,C 90.000,E1 259.577} C_DIS
LIN {X -0.057,Y -175.886,Z 1743.414,A 0.000,B 0.000,C 90.000,E1 254.519} C_DIS
LIN {X 0.049,Y -174.553,Z 1743.404,A 0.000,B 0.000,C 90.000,E1 252.779} C_DIS
LIN {X -0.019,Y -171.537,Z 1743.381,A 0.000,B 0.000,C 90.000,E1 248.518} C_DIS
LIN {X -0.025,Y -167.763,Z 1743.357,A 0.000,B 0.000,C 90.000,E1 244.204} C_DIS
LIN {X -0.083,Y -166.469,Z 1743.347,A 0.000,B 0.000,C 90.000,E1 242.487} C_DIS
LIN {X 0.053,Y -163.183,Z 1743.328,A 0.000,B 0.000,C 90.000,E1 238.948} C_DIS
LIN {X -0.032,Y -161.144,Z 1743.313,A 0.000,B 0.000,C 90.000,E1 236.342} C_DIS
LIN {X 0.004,Y -157.163,Z 1743.288,A 0.000,B 0.000,C 90.000,E1 231.904} C_DIS
LIN {X 0.027,Y -155.894,Z 1743.278,A 0.000,B 0.000,C 90.000,E1 230.114} C_DIS
LIN {X -0.015,Y -152.144,Z 1743.254,A 0.000,B 0.000,C 90.000,E1 225.648} C_DIS
LIN {X 0.005,Y -150.394,Z 1743.239,A 0.000,B 0.000,C 90.000,E1 222.933} C_DIS
LIN {X 0.029,Y -147.125,Z 1743.213,A 0.000,B 0.000,C 90.000,E1 218.382} C_DIS
LIN {X 0.020,Y -145.688,Z 1743.198,A 0.000,B 0.000,C 90.000,E1 215.644} C_DIS
LIN {X 0.017,Y -143.071,Z 1743.173,A 0.000,B 0.000,C 90.000,E1 211.052} C_DIS
LIN {X -0.051,Y -141.691,Z 1743.152,A 0.000,B 0.000,C 90.000,E1 207.385} C_DIS
LIN {X 0.003,Y -139.461,Z 1743.116,A 0.000,B 0.000,C 90.000,E1 200.865} C_DIS
LIN {X -0.028,Y -139.195,Z 1743.106,A 0.000,B 0.000,C 90.000,E1 199.014} C_DIS
LIN {X -0.010,Y -138.326,Z 1743.054,A 0.000,B 0.000,C 90.000,E1 189.670} C_DIS
LIN {X -0.005,Y -139.451,Z 1743.007,A 0.000,B 0.000,C 90.000,E1 181.260} C_DIS
LIN {X -0.066,Y -140.994,Z 1742.976,A 0.000,B 0.000,C 90.000,E1 175.698} C_DIS
LIN {X 0.025,Y -142.749,Z 1742.955,A 0.000,B 0.000,C 90.000,E1 171.951} C_DIS
LIN {X -0.019,Y -145.148,Z 1742.930,A 0.000,B 0.000,C 90.000,E1 167.353} C_DIS
LIN {X -0.025,Y -147.771,Z 1742.909,A 0.000,B 0.000,C 90.000,E1 163.685} C_DIS
LIN {X 0.054,Y -150.445,Z 1742.889,A 0.000,B 0.000,C 90.000,E1 160.007} C_DIS
LIN {X -0.012,Y -153.892,Z 1742.869,A 0.000,B 0.000,C 90.000,E1 156.410} C_DIS
LIN {X -0.018,Y -157.303,Z 1742.849,A 0.000,B 0.000,C 90.000,E1 152.820} C_DIS
LIN {X 0.001,Y -161.487,Z 1742.829,A 0.000,B 0.000,C 90.000,E1 149.253} C_DIS
LIN {X 0.017,Y -165.687,Z 1742.810,A 0.000,B 0.000,C 90.000,E1 145.722} C_DIS
LIN {X -0.096,Y -170.628,Z 1742.790,A 0.000,B 0.000,C 90.000,E1 142.271} C_DIS
LIN {X 0.057,Y -175.504,Z 1742.771,A 0.000,B 0.000,C 90.000,E1 138.771} C_DIS
LIN {X -0.077,Y -181.126,Z 1742.752,A 0.000,B 0.000,C 90.000,E1 135.405} C_DIS
LIN {X 0.050,Y -186.574,Z 1742.733,A 0.000,B 0.000,C 90.000,E1 132.000} C_DIS
LIN {X 0.000,Y -191.186,Z 1742.720,A 0.000,B 0.000,C 90.000,E1 129.519} C_DIS
LIN {X 0.046,Y -196.995,Z 1742.701,A 0.000,B 0.000,C 90.000,E1 126.217} C_DIS
LIN {X -0.036,Y -200.264,Z 1742.692,A 0.000,B 0.000,C 90.000,E1 124.612} C_DIS
LIN {X -0.042,Y -207.755,Z 1742.670,A 0.000,B 0.000,C 90.000,E1 120.590} C_DIS
LIN {X -0.115,Y -210.249,Z 1742.663,A 0.000,B 0.000,C 90.000,E1 119.411} C_DIS
LIN {X 0.048,Y -335.193,Z 1742.663,A 0.000,B 0.000,C 90.000,E1 119.361} C_DIS
LIN {X 0.154,Y -336.205,Z 1742.663,A 0.000,B 0.000,C 90.000,E1 119.333} C_DIS
LIN {X 0.112,Y -341.299,Z 1742.662,A 0.000,B 0.000,C 90.000,E1 119.155} C_DIS
LIN {X -0.065,Y -343.851,Z 1742.661,A 0.000,B 0.000,C 90.000,E1 118.999} C_DIS
LIN {X -0.019,Y -347.659,Z 1742.659,A 0.000,B 0.000,C 90.000,E1 118.565} C_DIS
LIN {X -0.102,Y -349.496,Z 1742.657,A 0.000,B 0.000,C 90.000,E1 118.281} C_DIS
LIN {X 0.050,Y -365.596,Z 1742.639,A 0.000,B 0.000,C 90.000,E1 114.951} C_DIS
LIN {X -0.131,Y -380.422,Z 1742.624,A 0.000,B 0.000,C 90.000,E1 112.333} C_DIS
LIN {X 0.154,Y -395.009,Z 1742.611,A 0.000,B 0.000,C 90.000,E1 109.993} C_DIS
LIN {X 0.037,Y -411.022,Z 1742.599,A 0.000,B 0.000,C 90.000,E1 107.764} C_DIS
LIN {X -0.212,Y -428.572,Z 1742.587,A 0.000,B 0.000,C 90.000,E1 105.607} C_DIS
LIN {X -0.137,Y -447.738,Z 1742.575,A 0.000,B 0.000,C 90.000,E1 103.467} C_DIS
LIN {X -0.136,Y -467.803,Z 1742.564,A 0.000,B 0.000,C 90.000,E1 101.478} C_DIS
LIN {X -0.163,Y -491.027,Z 1742.552,A 0.000,B 0.000,C 90.000,E1 99.434} C_DIS
LIN {X 0.138,Y -509.449,Z 1742.544,A 0.000,B 0.000,C 90.000,E1 97.936} C_DIS
LIN {X -0.074,Y -511.577,Z 1742.543,A 0.000,B 0.000,C 90.000,E1 97.757} C_DIS
LIN {X -0.116,Y -513.421,Z 1742.542,A 0.000,B 0.000,C 90.000,E1 97.530} C_DIS
LIN {X -0.089,Y -514.815,Z 1742.541,A 0.000,B 0.000,C 90.000,E1 97.296} C_DIS
LIN {X -0.232,Y -516.636,Z 1742.538,A 0.000,B 0.000,C 90.000,E1 96.834} C_DIS
LIN {X 0.147,Y -517.319,Z 1742.535,A 0.000,B 0.000,C 90.000,E1 96.315} C_DIS
LIN {X 0.021,Y -516.979,Z 1742.532,A 0.000,B 0.000,C 90.000,E1 95.853} C_DIS
LIN {X -0.102,Y -515.557,Z 1742.530,A 0.000,B 0.000,C 90.000,E1 95.391} C_DIS
LIN {X -0.188,Y -514.362,Z 1742.529,A 0.000,B 0.000,C 90.000,E1 95.163} C_DIS
LIN {X 0.190,Y -510.955,Z 1742.526,A 0.000,B 0.000,C 90.000,E1 94.645} C_DIS
LIN {X -0.217,Y -494.771,Z 1742.514,A 0.000,B 0.000,C 90.000,E1 92.522} C_DIS
LIN {X -0.057,Y -483.825,Z 1742.506,A 0.000,B 0.000,C 90.000,E1 91.031} C_DIS
LIN {X 0.007,Y -469.196,Z 1742.495,A 0.000,B 0.000,C 90.000,E1 89.026} C_DIS
LIN {X 0.194,Y -458.194,Z 1742.486,A 0.000,B 0.000,C 90.000,E1 87.478} C_DIS
LIN {X -0.035,Y -445.335,Z 1742.476,A 0.000,B 0.000,C 90.000,E1 85.698} C_DIS
LIN {X -0.031,Y -432.572,Z 1742.466,A 0.000,B 0.000,C 90.000,E1 83.856} C_DIS
LIN {X -0.141,Y -418.248,Z 1742.454,A 0.000,B 0.000,C 90.000,E1 81.724} C_DIS
LIN {X 0.214,Y -401.035,Z 1742.439,A 0.000,B 0.000,C 90.000,E1 78.926} C_DIS
LIN {X 0.138,Y -384.873,Z 1742.423,A 0.000,B 0.000,C 90.000,E1 76.117} C_DIS
LIN {X -0.126,Y -372.446,Z 1742.410,A 0.000,B 0.000,C 90.000,E1 73.850} C_DIS
LIN {X 0.087,Y -358.799,Z 1742.396,A 0.000,B 0.000,C 90.000,E1 71.167} C_DIS
LIN {X 0.091,Y -342.887,Z 1742.377,A 0.000,B 0.000,C 90.000,E1 67.847} C_DIS
LIN {X -0.072,Y -333.211,Z 1742.365,A 0.000,B 0.000,C 90.000,E1 65.717} C_DIS
LIN {X 0.045,Y -320.885,Z 1742.349,A 0.000,B 0.000,C 90.000,E1 62.871} C_DIS
LIN {X -0.063,Y -312.756,Z 1742.339,A 0.000,B 0.000,C 90.000,E1 60.973} C_DIS
LIN {X 0.103,Y -304.318,Z 1742.328,A 0.000,B 0.000,C 90.000,E1 58.997} C_DIS
LIN {X 0.010,Y -294.423,Z 1742.315,A 0.000,B 0.000,C 90.000,E1 56.707} C_DIS
LIN {X 0.024,Y -284.473,Z 1742.302,A 0.000,B 0.000,C 90.000,E1 54.356} C_DIS
LIN {X 0.025,Y -273.240,Z 1742.287,A 0.000,B 0.000,C 90.000,E1 51.618} C_DIS
LIN {X 0.019,Y -263.520,Z 1742.273,A 0.000,B 0.000,C 90.000,E1 49.175} C_DIS
LIN {X -0.031,Y -252.815,Z 1742.257,A 0.000,B 0.000,C 90.000,E1 46.338} C_DIS
LIN {X 0.013,Y -242.424,Z 1742.241,A 0.000,B 0.000,C 90.000,E1 43.419} C_DIS
LIN {X -0.053,Y -231.332,Z 1742.223,A 0.000,B 0.000,C 90.000,E1 40.092} C_DIS
LIN {X 0.046,Y -222.106,Z 1742.206,A 0.000,B 0.000,C 90.000,E1 37.030} C_DIS
LIN {X -0.143,Y -213.694,Z 1742.189,A 0.000,B 0.000,C 90.000,E1 33.992} C_DIS
LIN {X 0.054,Y -206.068,Z 1742.171,A 0.000,B 0.000,C 90.000,E1 30.797} C_DIS
LIN {X -0.080,Y -199.169,Z 1742.153,A 0.000,B 0.000,C 90.000,E1 27.641} C_DIS
LIN {X -0.035,Y -193.004,Z 1742.135,A 0.000,B 0.000,C 90.000,E1 24.387} C_DIS
LIN {X -0.027,Y -187.496,Z 1742.117,A 0.000,B 0.000,C 90.000,E1 21.099} C_DIS
LIN {X 0.002,Y -182.799,Z 1742.099,A 0.000,B 0.000,C 90.000,E1 17.764} C_DIS
LIN {X -0.024,Y -178.882,Z 1742.080,A 0.000,B 0.000,C 90.000,E1 14.411} C_DIS
LIN {X 0.063,Y -175.102,Z 1742.056,A 0.000,B 0.000,C 90.000,E1 10.141} C_DIS
LIN {X -0.073,Y -171.896,Z 1742.028,A 0.000,B 0.000,C 90.000,E1 5.049} C_DIS
LIN {X -0.056,Y -169.922,Z 1741.988,A 0.000,B 0.000,C 90.000,E1 357.822} C_DIS
LIN {X -0.060,Y -170.241,Z 1741.945,A 0.000,B 0.000,C 90.000,E1 350.038} C_DIS
LIN {X 0.001,Y -172.168,Z 1741.911,A 0.000,B 0.000,C 90.000,E1 343.976} C_DIS
LIN {X -0.011,Y -175.243,Z 1741.882,A 0.000,B 0.000,C 90.000,E1 338.827} C_DIS
LIN {X 0.071,Y -178.853,Z 1741.859,A 0.000,B 0.000,C 90.000,E1 334.537} C_DIS
LIN {X -0.014,Y -182.312,Z 1741.840,A 0.000,B 0.000,C 90.000,E1 331.179} C_DIS
LIN {X 0.097,Y -186.697,Z 1741.821,A 0.000,B 0.000,C 90.000,E1 327.788} C_DIS
LIN {X 0.043,Y -191.948,Z 1741.803,A 0.000,B 0.000,C 90.000,E1 324.482} C_DIS
LIN {X -0.001,Y -196.585,Z 1741.789,A 0.000,B 0.000,C 90.000,E1 322.029} C_DIS
LIN {X 0.011,Y -201.936,Z 1741.776,A 0.000,B 0.000,C 90.000,E1 319.585} C_DIS
LIN {X -0.007,Y -209.004,Z 1741.760,A 0.000,B 0.000,C 90.000,E1 316.782} C_DIS
LIN {X -0.082,Y -215.892,Z 1741.747,A 0.000,B 0.000,C 90.000,E1 314.433} C_DIS
LIN {X 0.061,Y -222.419,Z 1741.736,A 0.000,B 0.000,C 90.000,E1 312.447} C_DIS
LIN {X -0.045,Y -231.418,Z 1741.723,A 0.000,B 0.000,C 90.000,E1 310.172} C_DIS
LIN {X -0.075,Y -238.225,Z 1741.715,A 0.000,B 0.000,C 90.000,E1 308.669} C_DIS
LIN {X 0.008,Y -249.590,Z 1741.702,A 0.000,B 0.000,C 90.000,E1 306.423} C_DIS
LIN {X -0.089,Y -264.322,Z 1741.688,A 0.000,B 0.000,C 90.000,E1 303.913} C_DIS
LIN {X 0.032,Y -282.831,Z 1741.673,A 0.000,B 0.000,C 90.000,E1 301.082} C_DIS
LIN {X 0.119,Y -302.820,Z 1741.658,A 0.000,B 0.000,C 90.000,E1 298.359} C_DIS
LIN {X -0.048,Y -321.213,Z 1741.645,A 0.000,B 0.000,C 90.000,E1 296.104} C_DIS
LIN {X -0.049,Y -334.462,Z 1741.636,A 0.000,B 0.000,C 90.000,E1 294.515} C_DIS
LIN {X 0.014,Y -347.596,Z 1741.628,A 0.000,B 0.000,C 90.000,E1 292.950} C_DIS
LIN {X 0.162,Y -357.720,Z 1741.621,A 0.000,B 0.000,C 90.000,E1 291.716} C_DIS
LIN {X -0.080,Y -367.500,Z 1741.614,A 0.000,B 0.000,C 90.000,E1 290.556} C_DIS
LIN {X 0.176,Y -374.409,Z 1741.609,A 0.000,B 0.000,C 90.000,E1 289.631} C_DIS
LIN {X 0.008,Y -380.575,Z 1741.604,A 0.000,B 0.000,C 90.000,E1 288.779} C_DIS
LIN {X 0.132,Y -384.234,Z 1741.601,A 0.000,B 0.000,C 90.000,E1 288.181} C_DIS
LIN {X 0.057,Y -388.807,Z 1741.596,A 0.000,B 0.000,C 90.000,E1 287.330} C_DIS
LIN {X 0.124,Y -391.292,Z 1741.593,A 0.000,B 0.000,C 90.000,E1 286.749} C_DIS
LIN {X 0.106,Y -394.246,Z 1741.588,A 0.000,B 0.000,C 90.000,E1 285.898} C_DIS
LIN {X -0.167,Y -395.842,Z 1741.585,A 0.000,B 0.000,C 90.000,E1 285.371} C_DIS
LIN {X 0.057,Y -397.081,Z 1741.582,A 0.000,B 0.000,C 90.000,E1 284.773} C_DIS
LIN {X -0.194,Y -397.913,Z 1741.579,A 0.000,B 0.000,C 90.000,E1 284.245} C_DIS
LIN {X 0.046,Y -398.425,Z 1741.576,A 0.000,B 0.000,C 90.000,E1 283.647} C_DIS
LIN {X -0.193,Y -398.583,Z 1741.573,A 0.000,B 0.000,C 90.000,E1 283.119} C_DIS
LIN {X -0.038,Y -398.307,Z 1741.570,A 0.000,B 0.000,C 90.000,E1 282.535} C_DIS
LIN {X 0.118,Y -397.612,Z 1741.567,A 0.000,B 0.000,C 90.000,E1 281.951} C_DIS
LIN {X -0.114,Y -396.401,Z 1741.563,A 0.000,B 0.000,C 90.000,E1 281.422} C_DIS
LIN {X 0.036,Y -394.678,Z 1741.560,A 0.000,B 0.000,C 90.000,E1 280.838} C_DIS
LIN {X 0.178,Y -392.332,Z 1741.557,A 0.000,B 0.000,C 90.000,E1 280.254} C_DIS
LIN {X -0.085,Y -389.409,Z 1741.554,A 0.000,B 0.000,C 90.000,E1 279.726} C_DIS
LIN {X 0.041,Y -382.650,Z 1741.548,A 0.000,B 0.000,C 90.000,E1 278.568} C_DIS
LIN {X -0.028,Y -376.899,Z 1741.542,A 0.000,B 0.000,C 90.000,E1 277.466} C_DIS
LIN {X -0.055,Y -373.449,Z 1741.538,A 0.000,B 0.000,C 90.000,E1 276.891} C_DIS
LIN {X -0.099,Y -369.342,Z 1741.535,A 0.000,B 0.000,C 90.000,E1 276.315} C_DIS
LIN {X -0.164,Y -364.453,Z 1741.532,A 0.000,B 0.000,C 90.000,E1 275.739} C_DIS
LIN {X 0.105,Y -358.845,Z 1741.528,A 0.000,B 0.000,C 90.000,E1 275.106} C_DIS
LIN {X -0.112,Y -352.941,Z 1741.525,A 0.000,B 0.000,C 90.000,E1 274.588} C_DIS
LIN {X -0.126,Y -343.863,Z 1741.521,A 0.000,B 0.000,C 90.000,E1 273.841} C_DIS
LIN {X -0.125,Y -337.692,Z 1741.519,A 0.000,B 0.000,C 90.000,E1 273.383} C_DIS
LIN {X 0.082,Y -331.344,Z 1741.516,A 0.000,B 0.000,C 90.000,E1 272.922} C_DIS
LIN {X 0.138,Y -324.763,Z 1741.514,A 0.000,B 0.000,C 90.000,E1 272.522} C_DIS
LIN {X 0.095,Y -317.999,Z 1741.512,A 0.000,B 0.000,C 90.000,E1 272.178} C_DIS
LIN {X -0.006,Y -310.935,Z 1741.510,A 0.000,B 0.000,C 90.000,E1 271.892} C_DIS
LIN {X 0.136,Y -303.760,Z 1741.509,A 0.000,B 0.000,C 90.000,E1 271.604} C_DIS
LIN {X -0.033,Y -292.705,Z 1741.507,A 0.000,B 0.000,C 90.000,E1 271.318} C_DIS
LIN {X -0.036,Y -285.132,Z 1741.506,A 0.000,B 0.000,C 90.000,E1 271.146} C_DIS
LIN {X 0.065,Y -272.569,Z 1741.505,A 0.000,B 0.000,C 90.000,E1 270.917} C_DIS
LIN {X 0.120,Y -252.347,Z 1741.504,A 0.000,B 0.000,C 90.000,E1 270.688} C_DIS
LIN {X 0.004,Y -238.867,Z 1741.504,A 0.000,B 0.000,C 90.000,E1 270.630} C_DIS
LIN {X -0.033,Y -181.545,Z 1741.503,A 0.000,B 0.000,C 90.000,E1 270.630} C_DIS
LIN {X -0.064,Y -181.295,Z 1741.494,A 0.000,B 0.000,C 90.000,E1 268.912} C_DIS
LIN {X -0.015,Y -180.907,Z 1741.475,A 0.000,B 0.000,C 90.000,E1 265.527} C_DIS
LIN {X 0.042,Y -180.759,Z 1741.470,A 0.000,B 0.000,C 90.000,E1 264.666} C_DIS
LIN {X -0.065,Y -178.852,Z 1741.442,A 0.000,B 0.000,C 90.000,E1 259.634} C_DIS
LIN {X 0.006,Y -175.895,Z 1741.414,A 0.000,B 0.000,C 90.000,E1 254.519} C_DIS
LIN {X -0.055,Y -174.571,Z 1741.405,A 0.000,B 0.000,C 90.000,E1 252.834} C_DIS
LIN {X -0.019,Y -171.553,Z 1741.381,A 0.000,B 0.000,C 90.000,E1 248.539} C_DIS
LIN {X 0.036,Y -167.777,Z 1741.357,A 0.000,B 0.000,C 90.000,E1 244.204} C_DIS
LIN {X -0.023,Y -166.489,Z 1741.347,A 0.000,B 0.000,C 90.000,E1 242.487} C_DIS
LIN {X -0.026,Y -163.200,Z 1741.328,A 0.000,B 0.000,C 90.000,E1 238.997} C_DIS
LIN {X 0.028,Y -161.164,Z 1741.313,A 0.000,B 0.000,C 90.000,E1 236.342} C_DIS
LIN {X 0.064,Y -157.180,Z 1741.288,A 0.000,B 0.000,C 90.000,E1 231.904} C_DIS
LIN {X -0.014,Y -155.910,Z 1741.279,A 0.000,B 0.000,C 90.000,E1 230.150} C_DIS
LIN {X 0.043,Y -152.161,Z 1741.254,A 0.000,B 0.000,C 90.000,E1 225.648} C_DIS
LIN {X 0.063,Y -150.410,Z 1741.239,A 0.000,B 0.000,C 90.000,E1 222.933} C_DIS
LIN {X 0.085,Y -147.138,Z 1741.213,A 0.000,B 0.000,C 90.000,E1 218.382} C_DIS
LIN {X -0.010,Y -145.698,Z 1741.198,A 0.000,B 0.000,C 90.000,E1 215.678} C_DIS
LIN {X -0.001,Y -143.081,Z 1741.173,A 0.000,B 0.000,C 90.000,E1 211.082} C_DIS
LIN {X 0.004,Y -141.699,Z 1741.152,A 0.000,B 0.000,C 90.000,E1 207.385} C_DIS
LIN {X -0.073,Y -139.466,Z 1741.116,A 0.000,B 0.000,C 90.000,E1 200.918} C_DIS
LIN {X -0.019,Y -139.199,Z 1741.106,A 0.000,B 0.000,C 90.000,E1 199.033} C_DIS
LIN {X 0.045,Y -138.327,Z 1741.054,A 0.000,B 0.000,C 90.000,E1 189.670} C_DIS
LIN {X 0.049,Y -139.446,Z 1741.007,A 0.000,B 0.000,C 90.000,E1 181.260} C_DIS
LIN {X -0.010,Y -140.985,Z 1740.976,A 0.000,B 0.000,C 90.000,E1 175.698} C_DIS
LIN {X -0.061,Y -142.740,Z 1740.955,A 0.000,B 0.000,C 90.000,E1 172.008} C_DIS
LIN {X 0.038,Y -145.133,Z 1740.930,A 0.000,B 0.000,C 90.000,E1 167.353} C_DIS
LIN {X 0.031,Y -147.756,Z 1740.909,A 0.000,B 0.000,C 90.000,E1 163.685} C_DIS
LIN {X -0.030,Y -150.427,Z 1740.889,A 0.000,B 0.000,C 90.000,E1 160.061} C_DIS
LIN {X -0.015,Y -153.869,Z 1740.869,A 0.000,B 0.000,C 90.000,E1 156.433} C_DIS
LIN {X 0.042,Y -157.280,Z 1740.849,A 0.000,B 0.000,C 90.000,E1 152.820} C_DIS
LIN {X -0.021,Y -161.459,Z 1740.829,A 0.000,B 0.000,C 90.000,E1 149.282} C_DIS
LIN {X -0.015,Y -165.660,Z 1740.810,A 0.000,B 0.000,C 90.000,E1 145.754} C_DIS
LIN {X -0.033,Y -170.596,Z 1740.790,A 0.000,B 0.000,C 90.000,E1 142.271} C_DIS
LIN {X 0.005,Y -175.472,Z 1740.771,A 0.000,B 0.000,C 90.000,E1 138.809} C_DIS
LIN {X -0.011,Y -181.095,Z 1740.752,A 0.000,B 0.000,C 90.000,E1 135.405} C_DIS
LIN {X -0.022,Y -186.538,Z 1740.734,A 0.000,B 0.000,C 90.000,E1 132.043} C_DIS
LIN {X -0.081,Y -191.154,Z 1740.720,A 0.000,B 0.000,C 90.000,E1 129.564} C_DIS
LIN {X -0.003,Y -196.957,Z 1740.701,A 0.000,B 0.000,C 90.000,E1 126.251} C_DIS
LIN {X 0.033,Y -200.222,Z 1740.692,A 0.000,B 0.000,C 90.000,E1 124.612} C_DIS
LIN {X 0.028,Y -207.716,Z 1740.670,A 0.000,B 0.000,C 90.000,E1 120.590} C_DIS
LIN {X -0.008,Y -210.193,Z 1740.663,A 0.000,B 0.000,C 90.000,E1 119.411} C_DIS
LIN {X -0.072,Y -335.021,Z 1740.663,A 0.000,B 0.000,C 90.000,E1 119.411} C_DIS
LIN {X -0.191,Y -336.648,Z 1740.663,A 0.000,B 0.000,C 90.000,E1 119.411} C_DIS
LIN {X -0.072,Y -341.312,Z 1740.662,A 0.000,B 0.000,C 90.000,E1 119.205} C_DIS
LIN {X 0.050,Y -343.813,Z 1740.661,A 0.000,B 0.000,C 90.000,E1 118.999} C_DIS
LIN {X 0.053,Y -347.626,Z 1740.659,A 0.000,B 0.000,C 90.000,E1 118.565} C_DIS
LIN {X -0.049,Y -349.452,Z 1740.657,A 0.000,B 0.000,C 90.000,E1 118.281} C_DIS
LIN {X 0.083,Y -365.546,Z 1740.639,A 0.000,B 0.000,C 90.000,E1 114.951} C_DIS
LIN {X -0.096,Y -380.368,Z 1740.624,A 0.000,B 0.000,C 90.000,E1 112.333} C_DIS
LIN {X 0.188,Y -394.952,Z 1740.611,A 0.000,B 0.000,C 90.000,E1 109.993} C_DIS
LIN {X 0.070,Y -410.962,Z 1740.599,A 0.000,B 0.000,C 90.000,E1 107.764} C_DIS
LIN {X -0.180,Y -428.509,Z 1740.587,A 0.000,B 0.000,C 90.000,E1 105.607} C_DIS
LIN {X -0.104,Y -447.671,Z 1740.575,A 0.000,B 0.000,C 90.000,E1 103.467} C_DIS
LIN {X -0.106,Y -467.736,Z 1740.564,A 0.000,B 0.000,C 90.000,E1 101.478} C_DIS
LIN {X -0.136,Y -490.957,Z 1740.552,A 0.000,B 0.000,C 90.000,E1 99.434} C_DIS
LIN {X 0.163,Y -509.363,Z 1740.544,A 0.000,B 0.000,C 90.000,E1 97.936} C_DIS
LIN {X -0.049,Y -511.450,Z 1740.543,A 0.000,B 0.000,C 90.000,E1 97.757} C_DIS
LIN {X -0.114,Y -513.281,Z 1740.542,A 0.000,B 0.000,C 90.000,E1 97.530} C_DIS
LIN {X -0.112,Y -514.658,Z 1740.540,A 0.000,B 0.000,C 90.000,E1 97.296} C_DIS
LIN {X 0.257,Y -516.426,Z 1740.538,A 0.000,B 0.000,C 90.000,E1 96.777} C_DIS
LIN {X 0.121,Y -517.067,Z 1740.535,A 0.000,B 0.000,C 90.000,E1 96.315} C_DIS
LIN {X -0.006,Y -516.685,Z 1740.532,A 0.000,B 0.000,C 90.000,E1 95.853} C_DIS
LIN {X -0.129,Y -515.217,Z 1740.530,A 0.000,B 0.000,C 90.000,E1 95.391} C_DIS
LIN {X -0.216,Y -513.993,Z 1740.529,A 0.000,B 0.000,C 90.000,E1 95.163} C_DIS
LIN {X 0.069,Y -508.750,Z 1740.525,A 0.000,B 0.000,C 90.000,E1 94.416} C_DIS
LIN {X 0.240,Y -494.375,Z 1740.514,A 0.000,B 0.000,C 90.000,E1 92.465} C_DIS
LIN {X -0.101,Y -483.416,Z 1740.506,A 0.000,B 0.000,C 90.000,E1 91.031} C_DIS
LIN {X -0.044,Y -468.803,Z 1740.495,A 0.000,B 0.000,C 90.000,E1 89.026} C_DIS
LIN {X -0.085,Y -455.979,Z 1740.485,A 0.000,B 0.000,C 90.000,E1 87.249} C_DIS
LIN {X -0.132,Y -441.288,Z 1740.473,A 0.000,B 0.000,C 90.000,E1 85.179} C_DIS
LIN {X -0.080,Y -426.733,Z 1740.461,A 0.000,B 0.000,C 90.000,E1 83.053} C_DIS
LIN {X 0.200,Y -412.535,Z 1740.449,A 0.000,B 0.000,C 90.000,E1 80.849} C_DIS
LIN {X -0.008,Y -394.026,Z 1740.432,A 0.000,B 0.000,C 90.000,E1 77.825} C_DIS
LIN {X -0.136,Y -379.735,Z 1740.418,A 0.000,B 0.000,C 90.000,E1 75.283} C_DIS
LIN {X -0.152,Y -367.391,Z 1740.405,A 0.000,B 0.000,C 90.000,E1 72.960} C_DIS
LIN {X 0.148,Y -353.862,Z 1740.390,A 0.000,B 0.000,C 90.000,E1 70.242} C_DIS
LIN {X -0.006,Y -338.259,Z 1740.372,A 0.000,B 0.000,C 90.000,E1 66.922} C_DIS
LIN {X 0.175,Y -328.533,Z 1740.360,A 0.000,B 0.000,C 90.000,E1 64.717} C_DIS
LIN {X -0.072,Y -317.662,Z 1740.346,A 0.000,B 0.000,C 90.000,E1 62.231} C_DIS
LIN {X 0.032,Y -309.435,Z 1740.335,A 0.000,B 0.000,C 90.000,E1 60.284} C_DIS
LIN {X 0.045,Y -299.572,Z 1740.322,A 0.000,B 0.000,C 90.000,E1 57.995} C_DIS
LIN {X 0.017,Y -291.115,Z 1740.311,A 0.000,B 0.000,C 90.000,E1 56.008} C_DIS
LIN {X 0.126,Y -281.146,Z 1740.298,A 0.000,B 0.000,C 90.000,E1 53.623} C_DIS
LIN {X -0.045,Y -271.412,Z 1740.285,A 0.000,B 0.000,C 90.000,E1 51.251} C_DIS
LIN {X -0.056,Y -260.355,Z 1740.269,A 0.000,B 0.000,C 90.000,E1 48.447} C_DIS
LIN {X 0.009,Y -249.722,Z 1740.253,A 0.000,B 0.000,C 90.000,E1 45.567} C_DIS
LIN {X 0.142,Y -239.407,Z 1740.237,A 0.000,B 0.000,C 90.000,E1 42.609} C_DIS
LIN {X 0.007,Y -228.529,Z 1740.218,A 0.000,B 0.000,C 90.000,E1 39.277} C_DIS
LIN {X 0.033,Y -219.496,Z 1740.201,A 0.000,B 0.000,C 90.000,E1 36.217} C_DIS
LIN {X 0.130,Y -211.335,Z 1740.184,A 0.000,B 0.000,C 90.000,E1 33.086} C_DIS
LIN {X 0.046,Y -203.946,Z 1740.167,A 0.000,B 0.000,C 90.000,E1 29.951} C_DIS
LIN {X 0.039,Y -197.253,Z 1740.149,A 0.000,B 0.000,C 90.000,E1 26.744} C_DIS
LIN {X -0.047,Y -191.288,Z 1740.131,A 0.000,B 0.000,C 90.000,E1 23.515} C_DIS
LIN {X 0.028,Y -186.021,Z 1740.112,A 0.000,B 0.000,C 90.000,E1 20.194} C_DIS
LIN {X 0.022,Y -181.540,Z 1740.094,A 0.000,B 0.000,C 90.000,E1 16.858} C_DIS
LIN {X 0.045,Y -177.829,Z 1740.075,A 0.000,B 0.000,C 90.000,E1 13.480} C_DIS
LIN {X -0.067,Y -174.301,Z 1740.051,A 0.000,B 0.000,C 90.000,E1 9.265} C_DIS
LIN {X 0.071,Y -171.300,Z 1740.023,A 0.000,B 0.000,C 90.000,E1 4.073} C_DIS
LIN {X 0.067,Y -169.590,Z 1739.973,A 0.000,B 0.000,C 90.000,E1 355.184} C_DIS
LIN {X -0.095,Y -171.012,Z 1739.925,A 0.000,B 0.000,C 90.000,E1 346.589} C_DIS
LIN {X -0.042,Y -173.359,Z 1739.897,A 0.000,B 0.000,C 90.000,E1 341.402} C_DIS
LIN {X 0.007,Y -176.459,Z 1739.873,A 0.000,B 0.000,C 90.000,E1 337.102} C_DIS
LIN {X -0.055,Y -180.381,Z 1739.849,A 0.000,B 0.000,C 90.000,E1 332.871} C_DIS
LIN {X 0.073,Y -184.327,Z 1739.830,A 0.000,B 0.000,C 90.000,E1 329.459} C_DIS
LIN {X 0.018,Y -189.176,Z 1739.812,A 0.000,B 0.000,C 90.000,E1 326.135} C_DIS
LIN {X -0.024,Y -194.976,Z 1739.794,A 0.000,B 0.000,C 90.000,E1 322.844} C_DIS
LIN {X 0.110,Y -200.145,Z 1739.780,A 0.000,B 0.000,C 90.000,E1 320.356} C_DIS
LIN {X 0.069,Y -208.070,Z 1739.762,A 0.000,B 0.000,C 90.000,E1 317.148} C_DIS
LIN {X -0.121,Y -216.086,Z 1739.747,A 0.000,B 0.000,C 90.000,E1 314.433} C_DIS
LIN {X 0.024,Y -222.637,Z 1739.736,A 0.000,B 0.000,C 90.000,E1 312.447} C_DIS
LIN {X -0.079,Y -231.637,Z 1739.723,A 0.000,B 0.000,C 90.000,E1 310.172} C_DIS
LIN {X 0.053,Y -240.233,Z 1739.713,A 0.000,B 0.000,C 90.000,E1 308.257} C_DIS
LIN {X -0.166,Y -251.766,Z 1739.700,A 0.000,B 0.000,C 90.000,E1 306.091} C_DIS
LIN {X 0.146,Y -266.739,Z 1739.686,A 0.000,B 0.000,C 90.000,E1 303.499} C_DIS
LIN {X 0.104,Y -285.459,Z 1739.671,A 0.000,B 0.000,C 90.000,E1 300.718} C_DIS
LIN {X 0.099,Y -303.061,Z 1739.658,A 0.000,B 0.000,C 90.000,E1 298.359} C_DIS
LIN {X -0.081,Y -321.480,Z 1739.645,A 0.000,B 0.000,C 90.000,E1 296.104} C_DIS
LIN {X 0.031,Y -334.554,Z 1739.636,A 0.000,B 0.000,C 90.000,E1 294.515} C_DIS
LIN {X 0.109,Y -347.680,Z 1739.628,A 0.000,B 0.000,C 90.000,E1 292.950} C_DIS
LIN {X 0.041,Y -357.637,Z 1739.621,A 0.000,B 0.000,C 90.000,E1 291.770} C_DIS
LIN {X 0.137,Y -367.429,Z 1739.614,A 0.000,B 0.000,C 90.000,E1 290.556} C_DIS
LIN {X 0.043,Y -374.362,Z 1739.609,A 0.000,B 0.000,C 90.000,E1 289.685} C_DIS
LIN {X 0.122,Y -378.628,Z 1739.606,A 0.000,B 0.000,C 90.000,E1 289.087} C_DIS
LIN {X -0.129,Y -382.479,Z 1739.603,A 0.000,B 0.000,C 90.000,E1 288.544} C_DIS
LIN {X 0.007,Y -385.929,Z 1739.600,A 0.000,B 0.000,C 90.000,E1 287.946} C_DIS
LIN {X -0.202,Y -388.892,Z 1739.597,A 0.000,B 0.000,C 90.000,E1 287.402} C_DIS
LIN {X 0.132,Y -392.515,Z 1739.592,A 0.000,B 0.000,C 90.000,E1 286.496} C_DIS
LIN {X -0.039,Y -394.421,Z 1739.589,A 0.000,B 0.000,C 90.000,E1 285.953} C_DIS
LIN {X 0.067,Y -396.035,Z 1739.585,A 0.000,B 0.000,C 90.000,E1 285.371} C_DIS
LIN {X -0.090,Y -397.249,Z 1739.582,A 0.000,B 0.000,C 90.000,E1 284.828} C_DIS
LIN {X 0.044,Y -398.107,Z 1739.579,A 0.000,B 0.000,C 90.000,E1 284.245} C_DIS
LIN {X -0.102,Y -398.663,Z 1739.576,A 0.000,B 0.000,C 90.000,E1 283.703} C_DIS
LIN {X 0.048,Y -398.819,Z 1739.573,A 0.000,B 0.000,C 90.000,E1 283.119} C_DIS
LIN {X -0.185,Y -398.568,Z 1739.570,A 0.000,B 0.000,C 90.000,E1 282.591} C_DIS
LIN {X -0.028,Y -397.954,Z 1739.567,A 0.000,B 0.000,C 90.000,E1 282.007} C_DIS
LIN {X 0.129,Y -396.747,Z 1739.564,A 0.000,B 0.000,C 90.000,E1 281.422} C_DIS
LIN {X -0.107,Y -395.067,Z 1739.560,A 0.000,B 0.000,C 90.000,E1 280.894} C_DIS
LIN {X 0.037,Y -392.771,Z 1739.557,A 0.000,B 0.000,C 90.000,E1 280.310} C_DIS
LIN {X 0.161,Y -389.880,Z 1739.554,A 0.000,B 0.000,C 90.000,E1 279.726} C_DIS
LIN {X -0.035,Y -381.687,Z 1739.546,A 0.000,B 0.000,C 90.000,E1 278.341} C_DIS
LIN {X 0.068,Y -377.210,Z 1739.542,A 0.000,B 0.000,C 90.000,E1 277.473} C_DIS
LIN {X 0.090,Y -373.711,Z 1739.538,A 0.000,B 0.000,C 90.000,E1 276.891} C_DIS
LIN {X 0.046,Y -369.591,Z 1739.535,A 0.000,B 0.000,C 90.000,E1 276.315} C_DIS
LIN {X -0.019,Y -364.729,Z 1739.532,A 0.000,B 0.000,C 90.000,E1 275.739} C_DIS
LIN {X -0.108,Y -359.106,Z 1739.529,A 0.000,B 0.000,C 90.000,E1 275.163} C_DIS
LIN {X 0.010,Y -353.153,Z 1739.526,A 0.000,B 0.000,C 90.000,E1 274.588} C_DIS
LIN {X 0.036,Y -347.130,Z 1739.523,A 0.000,B 0.000,C 90.000,E1 274.073} C_DIS
LIN {X 0.014,Y -337.958,Z 1739.519,A 0.000,B 0.000,C 90.000,E1 273.383} C_DIS
LIN {X -0.109,Y -331.616,Z 1739.516,A 0.000,B 0.000,C 90.000,E1 272.980} C_DIS
LIN {X -0.051,Y -324.977,Z 1739.514,A 0.000,B 0.000,C 90.000,E1 272.579} C_DIS
LIN {X -0.089,Y -318.238,Z 1739.512,A 0.000,B 0.000,C 90.000,E1 272.236} C_DIS
LIN {X -0.015,Y -307.521,Z 1739.510,A 0.000,B 0.000,C 90.000,E1 271.776} C_DIS
